KUKA KRL program: EPS_2_25369_MH2A_A_20251128065456.src

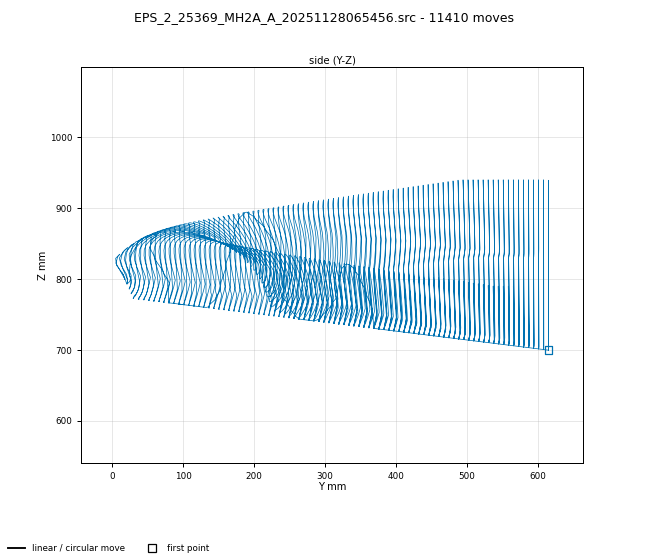
[picture p0: tool path of EPS_2_25369_MH2A_A_20251128065456.src, 11410 of 11412 moves have a stored position in this frame; points joined in program order, loops and branches not executed]
&ACCESS RVP
&REL 4
&COMMENT QRS 19112012
&PARAM EDITMASK = *
DEF PART()
EXT BAS (BAS_COMMAND :IN,REAL :IN )
INT I
BAS (#INITMOV,0 )

;KUKA QRS Post kuka4.cps  Date:22-06-2017 !

File_ID=2932

QRS_PRE_INIT()

;Init var - Until changes are made in qrs_pre_init
Outlet_Square_prg=0
Inlet_1_Square_prg=0
Inlet_2_Square_prg=0
Inlet_3_Square_prg=0
Inlet_4_Square_prg=0
Inlet_5_Square_prg=0

Outlet_1={X 0.000, Y 493.160, Z 839.500, B 0.000, E1 0.000 }
Inlet_1={X 0.000, Y 536.730, Z 239.500, B 0.000, E1 242.000 }
Outlet_1_type=201
Inlet_1_type=201
;QRS#1=Sidecore dimensions
;QRS#2=200-8" PVC SDR 35
;QRS#3=200-8" PVC SDR 35
;QRS#4=
;QRS#5=
;QRS#6=
;QRS#7=
;QRS#8=
;QRS#9=12-08 PSX
;QRS#10=12-08 PSX
;QRS#11=
;QRS#12=
;QRS#13=
;QRS#14=
;QRS#15=
;QRS#16=1220x127x1219 4'
;QRS#17=EPS Height
;QRS#18=940
;QRS#19=*
;QRS#20= UPDATED VERSION 22-06-2017
;QRS#21=*
Outlet_Square=0100
Inlet_1_Square=0100
Inlet_2_Square=0
Inlet_3_Square=0
Inlet_4_Square=0
Inlet_5_Square=0
Mill_Square=1
Outlet_Square_Prg=204
Inlet_1_Square_prg=204

QRS_INIT()

$ADVANCE=5

; T1
PTP {E1 173.443,E2 173.443}
PTP {X 0,Y 615.465,A -85,B 0,C 180,E1 173.443,E2 173.443,E3 0,E4 0,E5 0,E6 0}
QRS_SPEED_INIT()
LIN {X 0,Y 615.465,Z 699.696,A -85,B 0,C 180,E1 173.443,E2 173.443,E3 0,E4 0,E5 0,E6 0} C_VEL
LIN {X 0,Y 615.469,Z 699.697,A -85,B 0,C 180,E1 171.463,E2 171.463} C_VEL
LIN {X 0,Y 615.449,Z 699.694,A -85,B 0,C 180,E1 169.132,E2 169.132} C_VEL
LIN {X 0,Y 615.445,Z 699.691,A -85,B 0,C 180,E1 166.798,E2 166.798} C_VEL
LIN {X 0,Y 615.485,Z 699.687,A -85,B 0,C 180,E1 164.095,E2 164.095} C_VEL
LIN {X 0,Y 615.473,Z 699.698,A -85,B 0,C 180,E1 161.353,E2 161.353} C_VEL
LIN {X 0,Y 615.467,Z 699.698,A -85,B 0,C 180,E1 159.268,E2 159.268} C_VEL
LIN {X 0,Y 615.459,Z 699.697,A -85,B 0,C 180,E1 157.154,E2 157.154} C_VEL
LIN {X 0,Y 615.448,Z 699.697,A -85,B 0,C 180,E1 155.006,E2 155.006} C_VEL
LIN {X 0,Y 615.44,Z 699.696,A -85,B 0,C 180,E1 152.82,E2 152.82} C_VEL
LIN {X 0,Y 615.433,Z 699.695,A -85,B 0,C 180,E1 150.591,E2 150.591} C_VEL
LIN {X 0,Y 615.432,Z 699.694,A -85,B 0,C 180,E1 148.311,E2 148.311} C_VEL
LIN {X 0,Y 615.448,Z 699.692,A -85,B 0,C 180,E1 145.975,E2 145.975} C_VEL
LIN {X 0,Y 615.474,Z 699.699,A -85,B 0,C 180,E1 143.065,E2 143.065} C_VEL
LIN {X 0,Y 615.472,Z 699.697,A -85,B 0,C 180,E1 140.94,E2 140.94} C_VEL
LIN {X 0,Y 615.436,Z 699.696,A -85,B 0,C 180,E1 138.522,E2 138.522} C_VEL
LIN {X 0,Y 615.426,Z 699.695,A -85,B 0,C 180,E1 136.009,E2 136.009} C_VEL
LIN {X 0,Y 615.426,Z 699.695,A -85,B 0,C 180,E1 133.991,E2 133.991} C_VEL
LIN {X 0,Y 615.454,Z 699.695,A -85,B 0,C 180,E1 131.477,E2 131.477} C_VEL
LIN {X 0,Y 615.493,Z 699.698,A -85,B 0,C 180,E1 128.904,E2 128.904} C_VEL
LIN {X 0,Y 615.447,Z 699.695,A -85,B 0,C 180,E1 126.428,E2 126.428} C_VEL
LIN {X 0,Y 615.423,Z 699.696,A -85,B 0,C 180,E1 124.026,E2 124.026} C_VEL
LIN {X 0,Y 615.419,Z 699.697,A -85,B 0,C 180,E1 121.689,E2 121.689} C_VEL
LIN {X 0,Y 615.429,Z 699.698,A -85,B 0,C 180,E1 119.409,E2 119.409} C_VEL
LIN {X 0,Y 615.456,Z 699.7,A -85,B 0,C 180,E1 117.039,E2 117.039} C_VEL
LIN {X 0,Y 615.459,Z 699.694,A -85,B 0,C 180,E1 114.273,E2 114.273} C_VEL
LIN {X 0,Y 615.448,Z 699.694,A -85,B 0,C 180,E1 112.138,E2 112.138} C_VEL
LIN {X 0,Y 615.439,Z 699.695,A -85,B 0,C 180,E1 110.034,E2 110.034} C_VEL
LIN {X 0,Y 615.438,Z 699.695,A -85,B 0,C 180,E1 107.958,E2 107.958} C_VEL
LIN {X 0,Y 615.436,Z 699.695,A -85,B 0,C 180,E1 105.907,E2 105.907} C_VEL
LIN {X 0,Y 615.438,Z 699.695,A -85,B 0,C 180,E1 103.875,E2 103.875} C_VEL
LIN {X 0,Y 615.442,Z 699.694,A -85,B 0,C 180,E1 101.862,E2 101.862} C_VEL
LIN {X 0,Y 615.445,Z 699.694,A -85,B 0,C 180,E1 99.863,E2 99.863} C_VEL
LIN {X 0,Y 615.455,Z 699.692,A -85,B 0,C 180,E1 97.876,E2 97.876} C_VEL
LIN {X 0,Y 615.458,Z 699.693,A -85,B 0,C 180,E1 95.899,E2 95.899} C_VEL
LIN {X 0,Y 615.429,Z 699.694,A -85,B 0,C 180,E1 93.273,E2 93.273} C_VEL
LIN {X 0,Y 615.431,Z 699.694,A -85,B 0,C 180,E1 91.309,E2 91.309} C_VEL
LIN {X 0,Y 615.435,Z 699.693,A -85,B 0,C 180,E1 89.346,E2 89.346} C_VEL
LIN {X 0,Y 615.44,Z 699.692,A -85,B 0,C 180,E1 87.382,E2 87.382} C_VEL
LIN {X 0,Y 615.447,Z 699.691,A -85,B 0,C 180,E1 85.415,E2 85.415} C_VEL
LIN {X 0,Y 615.454,Z 699.69,A -85,B 0,C 180,E1 83.443,E2 83.443} C_VEL
LIN {X 0,Y 615.462,Z 699.689,A -85,B 0,C 180,E1 81.463,E2 81.463} C_VEL
LIN {X 0,Y 615.444,Z 699.691,A -85,B 0,C 180,E1 79.135,E2 79.135} C_VEL
LIN {X 0,Y 615.441,Z 699.693,A -85,B 0,C 180,E1 76.798,E2 76.798} C_VEL
LIN {X 0,Y 615.484,Z 699.701,A -85,B 0,C 180,E1 74.095,E2 74.095} C_VEL
LIN {X 0,Y 615.483,Z 699.685,A -85,B 0,C 180,E1 71.354,E2 71.354} C_VEL
LIN {X 0,Y 615.477,Z 699.686,A -85,B 0,C 180,E1 69.269,E2 69.269} C_VEL
LIN {X 0,Y 615.471,Z 699.686,A -85,B 0,C 180,E1 67.155,E2 67.155} C_VEL
LIN {X 0,Y 615.467,Z 699.686,A -85,B 0,C 180,E1 65.007,E2 65.007} C_VEL
LIN {X 0,Y 615.457,Z 699.688,A -85,B 0,C 180,E1 62.821,E2 62.821} C_VEL
LIN {X 0,Y 615.459,Z 699.695,A -85,B 0,C 180,E1 60.211,E2 60.211} C_VEL
LIN {X 0,Y 615.489,Z 699.695,A -85,B 0,C 180,E1 57.542,E2 57.542} C_VEL
LIN {X 0,Y 615.499,Z 699.684,A -85,B 0,C 180,E1 55.185,E2 55.185} C_VEL
LIN {X 0,Y 615.478,Z 699.683,A -85,B 0,C 180,E1 52.757,E2 52.757} C_VEL
LIN {X 0,Y 615.46,Z 699.69,A -85,B 0,C 180,E1 50.247,E2 50.247} C_VEL
LIN {X 0,Y 615.49,Z 699.699,A -85,B 0,C 180,E1 47.647,E2 47.647} C_VEL
LIN {X 0,Y 615.497,Z 699.683,A -85,B 0,C 180,E1 44.932,E2 44.932} C_VEL
LIN {X 0,Y 615.464,Z 699.69,A -85,B 0,C 180,E1 42.077,E2 42.077} C_VEL
LIN {X 0,Y 615.489,Z 699.696,A -85,B 0,C 180,E1 39.254,E2 39.254} C_VEL
LIN {X 0,Y 615.488,Z 714.003,A -85,B 0,C 180,E1 38.747,E2 38.747} C_VEL
LIN {X 0,Y 615.471,Z 726.147,A -85,B 0,C 180,E1 38.174,E2 38.174} C_VEL
LIN {X 0,Y 615.486,Z 736.877,A -85,B 0,C 180,E1 37.529,E2 37.529} C_VEL
LIN {X 0,Y 615.495,Z 746.56,A -85,B 0,C 180,E1 36.808,E2 36.808} C_VEL
LIN {X 0,Y 615.497,Z 755.612,A -85,B 0,C 180,E1 35.982,E2 35.982} C_VEL
LIN {X 0,Y 615.496,Z 764.246,A -85,B 0,C 180,E1 35.014,E2 35.014} C_VEL
LIN {X 0,Y 615.496,Z 771.392,A -85,B 0,C 180,E1 34.022,E2 34.022} C_VEL
LIN {X 0,Y 615.491,Z 775.986,A -85,B 0,C 180,E1 33.236,E2 33.236} C_VEL
LIN {X 0,Y 615.494,Z 781.677,A -85,B 0,C 180,E1 32.008,E2 32.008} C_VEL
LIN {X 0,Y 615.497,Z 785.306,A -85,B 0,C 180,E1 30.919,E2 30.919} C_VEL
LIN {X 0,Y 615.495,Z 787.813,A -85,B 0,C 180,E1 29.795,E2 29.795} C_VEL
LIN {X 0,Y 615.497,Z 789.275,A -85,B 0,C 180,E1 28.451,E2 28.451} C_VEL
LIN {X 0,Y 615.494,Z 789.086,A -85,B 0,C 180,E1 27.177,E2 27.177} C_VEL
LIN {X 0,Y 615.494,Z 788.342,A -85,B 0,C 180,E1 26.444,E2 26.444} C_VEL
LIN {X 0,Y 615.494,Z 786.748,A -85,B 0,C 180,E1 25.569,E2 25.569} C_VEL
LIN {X 0,Y 615.491,Z 784.237,A -85,B 0,C 180,E1 24.631,E2 24.631} C_VEL
LIN {X 0,Y 615.496,Z 780.239,A -85,B 0,C 180,E1 23.556,E2 23.556} C_VEL
LIN {X 0,Y 615.496,Z 775.556,A -85,B 0,C 180,E1 22.596,E2 22.596} C_VEL
LIN {X 0,Y 615.495,Z 769.504,A -85,B 0,C 180,E1 21.608,E2 21.608} C_VEL
LIN {X 0,Y 615.497,Z 761.465,A -85,B 0,C 180,E1 20.558,E2 20.558} C_VEL
LIN {X 0,Y 615.497,Z 753.124,A -85,B 0,C 180,E1 19.685,E2 19.685} C_VEL
LIN {X 0,Y 615.498,Z 742.968,A -85,B 0,C 180,E1 18.819,E2 18.819} C_VEL
LIN {X 0,Y 615.491,Z 732.83,A -85,B 0,C 180,E1 18.119,E2 18.119} C_VEL
LIN {X 0,Y 615.455,Z 722.15,A -85,B 0,C 180,E1 17.529,E2 17.529} C_VEL
LIN {X 0,Y 615.452,Z 710.214,A -85,B 0,C 180,E1 17.015,E2 17.015} C_VEL
LIN {X 0,Y 615.478,Z 699.698,A -85,B 0,C 180,E1 16.672,E2 16.672} C_VEL
LIN {X 0,Y 615.495,Z 699.683,A -85,B 0,C 180,E1 13.874,E2 13.874} C_VEL
LIN {X 0,Y 615.452,Z 699.69,A -85,B 0,C 180,E1 11.194,E2 11.194} C_VEL
LIN {X 0,Y 615.474,Z 699.698,A -85,B 0,C 180,E1 8.537,E2 8.537} C_VEL
LIN {X 0,Y 615.494,Z 699.688,A -85,B 0,C 180,E1 5.899,E2 5.899} C_VEL
LIN {X 0,Y 615.468,Z 699.685,A -85,B 0,C 180,E1 3.273,E2 3.273} C_VEL
LIN {X 0,Y 615.458,Z 699.694,A -85,B 0,C 180,E1 0.654,E2 0.654} C_VEL
LIN {X 0,Y 615.494,Z 699.697,A -85,B 0,C 180,E1 -1.963,E2 -1.963} C_VEL
LIN {X 0,Y 615.492,Z 699.682,A -85,B 0,C 180,E1 -4.584,E2 -4.584} C_VEL
LIN {X 0,Y 615.463,Z 699.688,A -85,B 0,C 180,E1 -7.216,E2 -7.216} C_VEL
LIN {X 0,Y 615.484,Z 699.698,A -85,B 0,C 180,E1 -9.862,E2 -9.862} C_VEL
LIN {X 0,Y 615.492,Z 699.686,A -85,B 0,C 180,E1 -12.53,E2 -12.53} C_VEL
LIN {X 0,Y 615.474,Z 699.684,A -85,B 0,C 180,E1 -15.226,E2 -15.226} C_VEL
LIN {X 0,Y 615.48,Z 699.697,A -85,B 0,C 180,E1 -17.957,E2 -17.957} C_VEL
LIN {X 0,Y 615.489,Z 699.686,A -85,B 0,C 180,E1 -20.731,E2 -20.731} C_VEL
LIN {X 0,Y 615.472,Z 699.686,A -85,B 0,C 180,E1 -23.557,E2 -23.557} C_VEL
LIN {X 0,Y 615.472,Z 699.688,A -85,B 0,C 180,E1 -25.716,E2 -25.716} C_VEL
LIN {X 0,Y 615.493,Z 699.698,A -85,B 0,C 180,E1 -28.45,E2 -28.45} C_VEL
LIN {X 0,Y 615.489,Z 699.683,A -85,B 0,C 180,E1 -31.086,E2 -31.086} C_VEL
LIN {X 0,Y 615.491,Z 699.68,A -85,B 0,C 180,E1 -33.534,E2 -33.534} C_VEL
LIN {X 0,Y 615.479,Z 699.686,A -85,B 0,C 180,E1 -35.832,E2 -35.832} C_VEL
LIN {X 0,Y 615.475,Z 699.69,A -85,B 0,C 180,E1 -38.07,E2 -38.07} C_VEL
LIN {X 0,Y 615.494,Z 699.7,A -85,B 0,C 180,E1 -40.606,E2 -40.606} C_VEL
LIN {X 0,Y 615.486,Z 699.685,A -85,B 0,C 180,E1 -43.245,E2 -43.245} C_VEL
LIN {X 0,Y 615.485,Z 699.684,A -85,B 0,C 180,E1 -46.003,E2 -46.003} C_VEL
LIN {X 0,Y 615.491,Z 699.695,A -85,B 0,C 180,E1 -48.905,E2 -48.905} C_VEL
LIN {X 0,Y 615.489,Z 699.691,A -85,B 0,C 180,E1 -51.095,E2 -51.095} C_VEL
LIN {X 0,Y 615.484,Z 699.683,A -85,B 0,C 180,E1 -53.575,E2 -53.575} C_VEL
LIN {X 0,Y 615.484,Z 699.799,A -85,B 0,C 180,E1 -54.356,E2 -54.356} C_VEL
LIN {X 0,Y 615.481,Z 713.626,A -85,B 0,C 180,E1 -57.153,E2 -57.153} C_VEL
LIN {X 0,Y 615.494,Z 727.321,A -85,B 0,C 180,E1 -59.84,E2 -59.84} C_VEL
LIN {X 0,Y 615.492,Z 741.016,A -85,B 0,C 180,E1 -62.454,E2 -62.454} C_VEL
LIN {X 0,Y 615.471,Z 754.706,A -85,B 0,C 180,E1 -65.007,E2 -65.007} C_VEL
LIN {X 0,Y 615.491,Z 769.177,A -85,B 0,C 180,E1 -67.654,E2 -67.654} C_VEL
LIN {X 0,Y 615.486,Z 784,A -85,B 0,C 180,E1 -70.315,E2 -70.315} C_VEL
LIN {X 0,Y 615.469,Z 799.609,A -85,B 0,C 180,E1 -73.071,E2 -73.071} C_VEL
LIN {X 0,Y 615.487,Z 815.037,A -85,B 0,C 180,E1 -75.761,E2 -75.761} C_VEL
LIN {X 0,Y 615.478,Z 829.932,A -85,B 0,C 180,E1 -78.327,E2 -78.327} C_VEL
LIN {X 0,Y 615.49,Z 843.234,A -85,B 0,C 180,E1 -78.557,E2 -78.557} C_VEL
LIN {X 0,Y 615.489,Z 856.372,A -85,B 0,C 180,E1 -78.923,E2 -78.923} C_VEL
LIN {X 0,Y 615.477,Z 868.148,A -85,B 0,C 180,E1 -79.384,E2 -79.384} C_VEL
LIN {X 0,Y 615.486,Z 879.573,A -85,B 0,C 180,E1 -79.972,E2 -79.972} C_VEL
LIN {X 0,Y 615.499,Z 891.019,A -85,B 0,C 180,E1 -80.718,E2 -80.718} C_VEL
LIN {X 0,Y 615.498,Z 900.256,A -85,B 0,C 180,E1 -81.463,E2 -81.463} C_VEL
LIN {X 0,Y 615.499,Z 908.652,A -85,B 0,C 180,E1 -82.29,E2 -82.29} C_VEL
LIN {X 0,Y 615.497,Z 916.69,A -85,B 0,C 180,E1 -83.259,E2 -83.259} C_VEL
LIN {X 0,Y 615.498,Z 922.422,A -85,B 0,C 180,E1 -84.101,E2 -84.101} C_VEL
LIN {X 0,Y 615.496,Z 927.872,A -85,B 0,C 180,E1 -85.087,E2 -85.087} C_VEL
LIN {X 0,Y 615.497,Z 932.141,A -85,B 0,C 180,E1 -86.071,E2 -86.071} C_VEL
LIN {X 0,Y 615.496,Z 934.398,A -85,B 0,C 180,E1 -86.727,E2 -86.727} C_VEL
LIN {X 0,Y 615.497,Z 936.233,A -85,B 0,C 180,E1 -87.382,E2 -87.382} C_VEL
LIN {X 0,Y 615.496,Z 937.608,A -85,B 0,C 180,E1 -88.037,E2 -88.037} C_VEL
LIN {X 0,Y 615.496,Z 939.173,A -85,B 0,C 180,E1 -89.346,E2 -89.346} C_VEL
LIN {X 0,Y 615.494,Z 939.389,A -85,B 0,C 180,E1 -90,E2 -90} C_VEL
LIN {X 0,Y 615.496,Z 938.58,A -85,B 0,C 180,E1 -91.309,E2 -91.309} C_VEL
LIN {X 0,Y 615.496,Z 937.608,A -85,B 0,C 180,E1 -91.963,E2 -91.963} C_VEL
LIN {X 0,Y 615.497,Z 936.233,A -85,B 0,C 180,E1 -92.618,E2 -92.618} C_VEL
LIN {X 0,Y 615.496,Z 933.35,A -85,B 0,C 180,E1 -93.601,E2 -93.601} C_VEL
LIN {X 0,Y 615.498,Z 929.442,A -85,B 0,C 180,E1 -94.584,E2 -94.584} C_VEL
LIN {X 0,Y 615.499,Z 924.405,A -85,B 0,C 180,E1 -95.57,E2 -95.57} C_VEL
LIN {X 0,Y 615.497,Z 917.869,A -85,B 0,C 180,E1 -96.583,E2 -96.583} C_VEL
LIN {X 0,Y 615.497,Z 910.133,A -85,B 0,C 180,E1 -97.545,E2 -97.545} C_VEL
LIN {X 0,Y 615.498,Z 902.045,A -85,B 0,C 180,E1 -98.371,E2 -98.371} C_VEL
LIN {X 0,Y 615.499,Z 892.168,A -85,B 0,C 180,E1 -99.199,E2 -99.199} C_VEL
LIN {X 0,Y 615.482,Z 880.983,A -85,B 0,C 180,E1 -99.945,E2 -99.945} C_VEL
LIN {X 0,Y 615.478,Z 870.024,A -85,B 0,C 180,E1 -100.527,E2 -100.527} C_VEL
LIN {X 0,Y 615.487,Z 857.564,A -85,B 0,C 180,E1 -101.037,E2 -101.037} C_VEL
LIN {X 0,Y 615.493,Z 845.064,A -85,B 0,C 180,E1 -101.401,E2 -101.401} C_VEL
LIN {X 0,Y 615.479,Z 831.469,A -85,B 0,C 180,E1 -101.652,E2 -101.652} C_VEL
LIN {X 0,Y 615.478,Z 829.797,A -85,B 0,C 180,E1 -101.694,E2 -101.694} C_VEL
LIN {X 0,Y 615.487,Z 815.037,A -85,B 0,C 180,E1 -104.239,E2 -104.239} C_VEL
LIN {X 0,Y 615.469,Z 799.61,A -85,B 0,C 180,E1 -106.929,E2 -106.929} C_VEL
LIN {X 0,Y 615.486,Z 784.001,A -85,B 0,C 180,E1 -109.685,E2 -109.685} C_VEL
LIN {X 0,Y 615.49,Z 767.803,A -85,B 0,C 180,E1 -112.595,E2 -112.595} C_VEL
LIN {X 0,Y 615.473,Z 753.141,A -85,B 0,C 180,E1 -115.282,E2 -115.282} C_VEL
LIN {X 0,Y 615.488,Z 739.06,A -85,B 0,C 180,E1 -117.915,E2 -117.915} C_VEL
LIN {X 0,Y 615.492,Z 725.365,A -85,B 0,C 180,E1 -120.539,E2 -120.539} C_VEL
LIN {X 0,Y 615.472,Z 711.67,A -85,B 0,C 180,E1 -123.237,E2 -123.237} C_VEL
LIN {X 0,Y 615.484,Z 699.687,A -85,B 0,C 180,E1 -125.671,E2 -125.671} C_VEL
LIN {X 0,Y 615.489,Z 699.681,A -85,B 0,C 180,E1 -128.069,E2 -128.069} C_VEL
LIN {X 0,Y 615.486,Z 699.684,A -85,B 0,C 180,E1 -130.607,E2 -130.607} C_VEL
LIN {X 0,Y 615.494,Z 699.699,A -85,B 0,C 180,E1 -133.244,E2 -133.244} C_VEL
LIN {X 0,Y 615.483,Z 699.685,A -85,B 0,C 180,E1 -136.003,E2 -136.003} C_VEL
LIN {X 0,Y 615.49,Z 699.686,A -85,B 0,C 180,E1 -138.905,E2 -138.905} C_VEL
LIN {X 0,Y 615.494,Z 699.689,A -85,B 0,C 180,E1 -141.096,E2 -141.096} C_VEL
LIN {X 0,Y 615.482,Z 699.7,A -85,B 0,C 180,E1 -143.575,E2 -143.575} C_VEL
LIN {X 0,Y 615.474,Z 699.691,A -85,B 0,C 180,E1 -145.977,E2 -145.977} C_VEL
LIN {X 0,Y 615.478,Z 699.685,A -85,B 0,C 180,E1 -148.314,E2 -148.314} C_VEL
LIN {X 0,Y 615.486,Z 699.681,A -85,B 0,C 180,E1 -150.594,E2 -150.594} C_VEL
LIN {X 0,Y 615.494,Z 699.697,A -85,B 0,C 180,E1 -153.556,E2 -153.556} C_VEL
LIN {X 0,Y 615.476,Z 699.695,A -85,B 0,C 180,E1 -155.995,E2 -155.995} C_VEL
LIN {X 0,Y 615.473,Z 699.685,A -85,B 0,C 180,E1 -158.568,E2 -158.568} C_VEL
LIN {X 0,Y 615.492,Z 699.688,A -85,B 0,C 180,E1 -161.395,E2 -161.395} C_VEL
LIN {X 0,Y 615.476,Z 699.696,A -85,B 0,C 180,E1 -164.095,E2 -164.095} C_VEL
LIN {X 0,Y 615.469,Z 699.685,A -85,B 0,C 180,E1 -166.798,E2 -166.798} C_VEL
LIN {X 0,Y 615.492,Z 699.686,A -85,B 0,C 180,E1 -169.473,E2 -169.473} C_VEL
LIN {X 0,Y 615.484,Z 699.698,A -85,B 0,C 180,E1 -172.124,E2 -172.124} C_VEL
LIN {X 0,Y 615.458,Z 699.689,A -85,B 0,C 180,E1 -174.759,E2 -174.759} C_VEL
LIN {X 0,Y 615.493,Z 699.682,A -85,B 0,C 180,E1 -177.382,E2 -177.382} C_VEL
LIN {X 0,Y 615.494,Z 699.697,A -85,B 0,C 180,E1 -180,E2 -180} C_VEL
LIN {X 0,Y 615.458,Z 699.694,A -85,B 0,C 180,E1 -182.618,E2 -182.618} C_VEL
LIN {X 0,Y 615.46,Z 699.687,A -85,B 0,C 180,E1 -185.242,E2 -185.242} C_VEL
LIN {X 0,Y 615.465,Z 699.696,A -85,B 0,C 180,E1 -186.557,E2 -186.557} C_VEL
LIN {X 0,Y 614.779,Z 699.837,A -85,B 0,C 180,E1 -187.103,E2 -187.103} C_VEL
LIN {X 0,Y 611.934,Z 700.259,A -85,B 0,C 180,E1 -187.99,E2 -187.99} C_VEL
LIN {X 0,Y 609.545,Z 700.565,A -85,B 0,C 180,E1 -188.702,E2 -188.702} C_VEL
LIN {X 0,Y 608.524,Z 700.679,A -85,B 0,C 180,E1 -189.252,E2 -189.252} C_VEL
LIN {X 0,Y 608.441,Z 700.688,A -85,B 0,C 180,E1 -189.438,E2 -189.438} C_VEL
LIN {X 0,Y 608.461,Z 700.691,A -85,B 0,C 180,E1 -192,E2 -192} C_VEL
LIN {X 0,Y 608.431,Z 700.694,A -85,B 0,C 180,E1 -194.722,E2 -194.722} C_VEL
LIN {X 0,Y 608.431,Z 700.694,A -85,B 0,C 180,E1 -196.785,E2 -196.785} C_VEL
LIN {X 0,Y 608.443,Z 700.692,A -85,B 0,C 180,E1 -198.87,E2 -198.87} C_VEL
LIN {X 0,Y 608.434,Z 700.692,A -85,B 0,C 180,E1 -200.982,E2 -200.982} C_VEL
LIN {X 0,Y 608.42,Z 700.693,A -85,B 0,C 180,E1 -203.125,E2 -203.125} C_VEL
LIN {X 0,Y 608.434,Z 700.689,A -85,B 0,C 180,E1 -205.713,E2 -205.713} C_VEL
LIN {X 0,Y 608.476,Z 700.695,A -85,B 0,C 180,E1 -208.62,E2 -208.62} C_VEL
LIN {X 0,Y 608.43,Z 700.691,A -85,B 0,C 180,E1 -211.319,E2 -211.319} C_VEL
LIN {X 0,Y 608.427,Z 700.69,A -85,B 0,C 180,E1 -213.728,E2 -213.728} C_VEL
LIN {X 0,Y 608.435,Z 700.69,A -85,B 0,C 180,E1 -216.093,E2 -216.093} C_VEL
LIN {X 0,Y 608.427,Z 700.697,A -85,B 0,C 180,E1 -218.592,E2 -218.592} C_VEL
LIN {X 0,Y 608.431,Z 700.692,A -85,B 0,C 180,E1 -221.339,E2 -221.339} C_VEL
LIN {X 0,Y 608.421,Z 700.691,A -85,B 0,C 180,E1 -223.874,E2 -223.874} C_VEL
LIN {X 0,Y 608.478,Z 700.69,A -85,B 0,C 180,E1 -226.691,E2 -226.691} C_VEL
LIN {X 0,Y 608.45,Z 700.696,A -85,B 0,C 180,E1 -228.823,E2 -228.823} C_VEL
LIN {X 0,Y 608.424,Z 700.691,A -85,B 0,C 180,E1 -231.765,E2 -231.765} C_VEL
LIN {X 0,Y 608.407,Z 700.693,A -85,B 0,C 180,E1 -233.96,E2 -233.96} C_VEL
LIN {X 0,Y 608.413,Z 700.692,A -85,B 0,C 180,E1 -236.326,E2 -236.326} C_VEL
LIN {X 0,Y 608.436,Z 700.693,A -85,B 0,C 180,E1 -238.735,E2 -238.735} C_VEL
LIN {X 0,Y 608.418,Z 700.693,A -85,B 0,C 180,E1 -241.732,E2 -241.732} C_VEL
LIN {X 0,Y 608.396,Z 700.694,A -85,B 0,C 180,E1 -244.295,E2 -244.295} C_VEL
LIN {X 0,Y 608.421,Z 700.695,A -85,B 0,C 180,E1 -246.875,E2 -246.875} C_VEL
LIN {X 0,Y 608.443,Z 700.692,A -85,B 0,C 180,E1 -249.725,E2 -249.725} C_VEL
LIN {X 0,Y 608.419,Z 700.694,A -85,B 0,C 180,E1 -251.827,E2 -251.827} C_VEL
LIN {X 0,Y 608.434,Z 700.692,A -85,B 0,C 180,E1 -253.905,E2 -253.905} C_VEL
LIN {X 0,Y 608.41,Z 700.692,A -85,B 0,C 180,E1 -256.642,E2 -256.642} C_VEL
LIN {X 0,Y 608.451,Z 700.695,A -85,B 0,C 180,E1 -259.35,E2 -259.35} C_VEL
LIN {X 0,Y 608.425,Z 700.693,A -85,B 0,C 180,E1 -262.032,E2 -262.032} C_VEL
LIN {X 0,Y 608.409,Z 700.692,A -85,B 0,C 180,E1 -264.698,E2 -264.698} C_VEL
LIN {X 0,Y 608.454,Z 700.692,A -85,B 0,C 180,E1 -267.352,E2 -267.352} C_VEL
LIN {X 0,Y 608.477,Z 700.689,A -85,B 0,C 180,E1 -270,E2 -270} C_VEL
LIN {X 0,Y 608.435,Z 700.689,A -85,B 0,C 180,E1 -272.648,E2 -272.648} C_VEL
LIN {X 0,Y 608.429,Z 700.693,A -85,B 0,C 180,E1 -275.302,E2 -275.302} C_VEL
LIN {X 0,Y 608.477,Z 700.693,A -85,B 0,C 180,E1 -277.967,E2 -277.967} C_VEL
LIN {X 0,Y 608.44,Z 700.689,A -85,B 0,C 180,E1 -280.65,E2 -280.65} C_VEL
LIN {X 0,Y 608.432,Z 700.691,A -85,B 0,C 180,E1 -283.357,E2 -283.357} C_VEL
LIN {X 0,Y 608.461,Z 700.695,A -85,B 0,C 180,E1 -286.094,E2 -286.094} C_VEL
LIN {X 0,Y 608.448,Z 700.687,A -85,B 0,C 180,E1 -288.87,E2 -288.87} C_VEL
LIN {X 0,Y 608.442,Z 700.688,A -85,B 0,C 180,E1 -290.982,E2 -290.982} C_VEL
LIN {X 0,Y 608.43,Z 700.689,A -85,B 0,C 180,E1 -293.125,E2 -293.125} C_VEL
LIN {X 0,Y 608.448,Z 700.691,A -85,B 0,C 180,E1 -295.715,E2 -295.715} C_VEL
LIN {X 0,Y 608.481,Z 700.687,A -85,B 0,C 180,E1 -298.621,E2 -298.621} C_VEL
LIN {X 0,Y 608.441,Z 700.688,A -85,B 0,C 180,E1 -301.318,E2 -301.318} C_VEL
LIN {X 0,Y 608.428,Z 700.692,A -85,B 0,C 180,E1 -303.728,E2 -303.728} C_VEL
LIN {X 0,Y 608.444,Z 700.695,A -85,B 0,C 180,E1 -306.093,E2 -306.093} C_VEL
LIN {X 0,Y 608.472,Z 700.692,A -85,B 0,C 180,E1 -308.588,E2 -308.588} C_VEL
LIN {X 0,Y 608.455,Z 700.686,A -85,B 0,C 180,E1 -311.341,E2 -311.341} C_VEL
LIN {X 0,Y 608.456,Z 700.688,A -85,B 0,C 180,E1 -313.871,E2 -313.871} C_VEL
LIN {X 0,Y 608.477,Z 700.692,A -85,B 0,C 180,E1 -316.691,E2 -316.691} C_VEL
LIN {X 0,Y 608.457,Z 700.686,A -85,B 0,C 180,E1 -319.697,E2 -319.697} C_VEL
LIN {X 0,Y 608.465,Z 700.696,A -85,B 0,C 180,E1 -320.654,E2 -320.654} C_VEL
LIN {X 0,Y 608.503,Z 713.389,A -85,B 0,C 180,E1 -321.096,E2 -321.096} C_VEL
LIN {X 0,Y 608.485,Z 724.662,A -85,B 0,C 180,E1 -321.619,E2 -321.619} C_VEL
LIN {X 0,Y 608.472,Z 736.703,A -85,B 0,C 180,E1 -322.335,E2 -322.335} C_VEL
LIN {X 0,Y 608.467,Z 746.782,A -85,B 0,C 180,E1 -323.086,E2 -323.086} C_VEL
LIN {X 0,Y 608.455,Z 756.207,A -85,B 0,C 180,E1 -323.954,E2 -323.954} C_VEL
LIN {X 0,Y 608.467,Z 764.899,A -85,B 0,C 180,E1 -324.938,E2 -324.938} C_VEL
LIN {X 0,Y 608.441,Z 771.955,A -85,B 0,C 180,E1 -325.928,E2 -325.928} C_VEL
LIN {X 0,Y 608.43,Z 778.577,A -85,B 0,C 180,E1 -327.119,E2 -327.119} C_VEL
LIN {X 0,Y 608.428,Z 783.503,A -85,B 0,C 180,E1 -328.293,E2 -328.293} C_VEL
LIN {X 0,Y 608.433,Z 786.942,A -85,B 0,C 180,E1 -329.453,E2 -329.453} C_VEL
LIN {X 0,Y 608.445,Z 788.467,A -85,B 0,C 180,E1 -330.219,E2 -330.219} C_VEL
LIN {X 0,Y 608.421,Z 789.788,A -85,B 0,C 180,E1 -331.39,E2 -331.39} C_VEL
LIN {X 0,Y 608.436,Z 789.717,A -85,B 0,C 180,E1 -332.801,E2 -332.801} C_VEL
LIN {X 0,Y 608.421,Z 788.314,A -85,B 0,C 180,E1 -333.963,E2 -333.963} C_VEL
LIN {X 0,Y 608.433,Z 785.822,A -85,B 0,C 180,E1 -335.063,E2 -335.063} C_VEL
LIN {X 0,Y 608.441,Z 782.175,A -85,B 0,C 180,E1 -336.154,E2 -336.154} C_VEL
LIN {X 0,Y 608.447,Z 777.282,A -85,B 0,C 180,E1 -337.235,E2 -337.235} C_VEL
LIN {X 0,Y 608.438,Z 770.991,A -85,B 0,C 180,E1 -338.307,E2 -338.307} C_VEL
LIN {X 0,Y 608.458,Z 763.49,A -85,B 0,C 180,E1 -339.325,E2 -339.325} C_VEL
LIN {X 0,Y 608.477,Z 755.053,A -85,B 0,C 180,E1 -340.254,E2 -340.254} C_VEL
LIN {X 0,Y 608.472,Z 745.197,A -85,B 0,C 180,E1 -341.131,E2 -341.131} C_VEL
LIN {X 0,Y 608.507,Z 734.234,A -85,B 0,C 180,E1 -341.917,E2 -341.917} C_VEL
LIN {X 0,Y 608.481,Z 723.664,A -85,B 0,C 180,E1 -342.524,E2 -342.524} C_VEL
LIN {X 0,Y 608.472,Z 712.168,A -85,B 0,C 180,E1 -343.043,E2 -343.043} C_VEL
LIN {X 0,Y 608.472,Z 700.695,A -85,B 0,C 180,E1 -343.446,E2 -343.446} C_VEL
LIN {X 0,Y 608.481,Z 700.687,A -85,B 0,C 180,E1 -345.98,E2 -345.98} C_VEL
LIN {X 0,Y 608.429,Z 700.69,A -85,B 0,C 180,E1 -348.675,E2 -348.675} C_VEL
LIN {X 0,Y 608.443,Z 700.694,A -85,B 0,C 180,E1 -351.364,E2 -351.364} C_VEL
LIN {X 0,Y 608.466,Z 700.69,A -85,B 0,C 180,E1 -354.033,E2 -354.033} C_VEL
LIN {X 0,Y 608.465,Z 700.685,A -85,B 0,C 180,E1 -356.689,E2 -356.689} C_VEL
LIN {X 0,Y 608.456,Z 700.69,A -85,B 0,C 180,E1 -359.338,E2 -359.338} C_VEL
LIN {X 0,Y 608.464,Z 700.694,A -85,B 0,C 180,E1 -361.986,E2 -361.986} C_VEL
LIN {X 0,Y 608.459,Z 700.687,A -85,B 0,C 180,E1 -364.638,E2 -364.638} C_VEL
LIN {X 0,Y 608.435,Z 700.69,A -85,B 0,C 180,E1 -367.3,E2 -367.3} C_VEL
LIN {X 0,Y 608.456,Z 700.697,A -85,B 0,C 180,E1 -369.977,E2 -369.977} C_VEL
LIN {X 0,Y 608.477,Z 700.685,A -85,B 0,C 180,E1 -372.677,E2 -372.677} C_VEL
LIN {X 0,Y 608.462,Z 700.686,A -85,B 0,C 180,E1 -375.406,E2 -375.406} C_VEL
LIN {X 0,Y 608.448,Z 700.699,A -85,B 0,C 180,E1 -378.172,E2 -378.172} C_VEL
LIN {X 0,Y 608.455,Z 700.687,A -85,B 0,C 180,E1 -380.982,E2 -380.982} C_VEL
LIN {X 0,Y 608.449,Z 700.687,A -85,B 0,C 180,E1 -383.124,E2 -383.124} C_VEL
LIN {X 0,Y 608.462,Z 700.688,A -85,B 0,C 180,E1 -385.718,E2 -385.718} C_VEL
LIN {X 0,Y 608.452,Z 700.697,A -85,B 0,C 180,E1 -388.267,E2 -388.267} C_VEL
LIN {X 0,Y 608.471,Z 700.693,A -85,B 0,C 180,E1 -390.545,E2 -390.545} C_VEL
LIN {X 0,Y 608.464,Z 700.689,A -85,B 0,C 180,E1 -392.879,E2 -392.879} C_VEL
LIN {X 0,Y 608.45,Z 700.687,A -85,B 0,C 180,E1 -395.277,E2 -395.277} C_VEL
LIN {X 0,Y 608.464,Z 700.686,A -85,B 0,C 180,E1 -397.747,E2 -397.747} C_VEL
LIN {X 0,Y 608.45,Z 700.694,A -85,B 0,C 180,E1 -400.328,E2 -400.328} C_VEL
LIN {X 0,Y 608.474,Z 700.685,A -85,B 0,C 180,E1 -403.309,E2 -403.309} C_VEL
LIN {X 0,Y 608.472,Z 700.687,A -85,B 0,C 180,E1 -406.13,E2 -406.13} C_VEL
LIN {X 0,Y 608.46,Z 700.696,A -85,B 0,C 180,E1 -408.823,E2 -408.823} C_VEL
LIN {X 0,Y 608.47,Z 700.685,A -85,B 0,C 180,E1 -411.76,E2 -411.76} C_VEL
LIN {X 0,Y 608.492,Z 700.74,A -85,B 0,C 180,E1 -414.08,E2 -414.08} C_VEL
LIN {X 0,Y 608.676,Z 706.578,A -85,B 0,C 180,E1 -415.302,E2 -415.302} C_VEL
LIN {X 0,Y 608.66,Z 719.495,A -85,B 0,C 180,E1 -417.917,E2 -417.917} C_VEL
LIN {X 0,Y 608.596,Z 733.19,A -85,B 0,C 180,E1 -420.608,E2 -420.608} C_VEL
LIN {X 0,Y 608.57,Z 746.885,A -85,B 0,C 180,E1 -423.231,E2 -423.231} C_VEL
LIN {X 0,Y 608.54,Z 760.792,A -85,B 0,C 180,E1 -425.835,E2 -425.835} C_VEL
LIN {X 0,Y 608.528,Z 776.232,A -85,B 0,C 180,E1 -428.666,E2 -428.666} C_VEL
LIN {X 0,Y 608.493,Z 792.297,A -85,B 0,C 180,E1 -431.555,E2 -431.555} C_VEL
LIN {X 0,Y 608.481,Z 807.534,A -85,B 0,C 180,E1 -434.251,E2 -434.251} C_VEL
LIN {X 0,Y 608.459,Z 823.186,A -85,B 0,C 180,E1 -436.983,E2 -436.983} C_VEL
LIN {X 0,Y 608.439,Z 830.156,A -85,B 0,C 180,E1 -438.19,E2 -438.19} C_VEL
LIN {X 0,Y 608.54,Z 844.261,A -85,B 0,C 180,E1 -438.445,E2 -438.445} C_VEL
LIN {X 0,Y 608.531,Z 856.957,A -85,B 0,C 180,E1 -438.81,E2 -438.81} C_VEL
LIN {X 0,Y 608.499,Z 868.679,A -85,B 0,C 180,E1 -439.279,E2 -439.279} C_VEL
LIN {X 0,Y 608.482,Z 879.753,A -85,B 0,C 180,E1 -439.855,E2 -439.855} C_VEL
LIN {X 0,Y 608.504,Z 891.25,A -85,B 0,C 180,E1 -440.611,E2 -440.611} C_VEL
LIN {X 0,Y 608.472,Z 900.535,A -85,B 0,C 180,E1 -441.364,E2 -441.364} C_VEL
LIN {X 0,Y 608.456,Z 908.988,A -85,B 0,C 180,E1 -442.2,E2 -442.2} C_VEL
LIN {X 0,Y 608.462,Z 917.234,A -85,B 0,C 180,E1 -443.201,E2 -443.201} C_VEL
LIN {X 0,Y 608.437,Z 923.876,A -85,B 0,C 180,E1 -444.199,E2 -444.199} C_VEL
LIN {X 0,Y 608.432,Z 929.95,A -85,B 0,C 180,E1 -445.362,E2 -445.362} C_VEL
LIN {X 0,Y 608.449,Z 933.896,A -85,B 0,C 180,E1 -446.358,E2 -446.358} C_VEL
LIN {X 0,Y 608.425,Z 936.809,A -85,B 0,C 180,E1 -447.352,E2 -447.352} C_VEL
LIN {X 0,Y 608.441,Z 938.201,A -85,B 0,C 180,E1 -448.014,E2 -448.014} C_VEL
LIN {X 0,Y 608.438,Z 939.783,A -85,B 0,C 180,E1 -449.338,E2 -449.338} C_VEL
LIN {X 0,Y 608.434,Z 940,A -85,B 0,C 180,E1 -450,E2 -450} C_VEL
LIN {X 0,Y 608.448,Z 939.184,A -85,B 0,C 180,E1 -451.324,E2 -451.324} C_VEL
LIN {X 0,Y 608.441,Z 938.201,A -85,B 0,C 180,E1 -451.986,E2 -451.986} C_VEL
LIN {X 0,Y 608.425,Z 936.809,A -85,B 0,C 180,E1 -452.648,E2 -452.648} C_VEL
LIN {X 0,Y 608.449,Z 933.896,A -85,B 0,C 180,E1 -453.642,E2 -453.642} C_VEL
LIN {X 0,Y 608.432,Z 929.95,A -85,B 0,C 180,E1 -454.638,E2 -454.638} C_VEL
LIN {X 0,Y 608.437,Z 923.877,A -85,B 0,C 180,E1 -455.801,E2 -455.801} C_VEL
LIN {X 0,Y 608.462,Z 917.235,A -85,B 0,C 180,E1 -456.799,E2 -456.799} C_VEL
LIN {X 0,Y 608.456,Z 908.989,A -85,B 0,C 180,E1 -457.8,E2 -457.8} C_VEL
LIN {X 0,Y 608.472,Z 900.536,A -85,B 0,C 180,E1 -458.636,E2 -458.636} C_VEL
LIN {X 0,Y 608.48,Z 890.091,A -85,B 0,C 180,E1 -459.473,E2 -459.473} C_VEL
LIN {X 0,Y 608.482,Z 879.755,A -85,B 0,C 180,E1 -460.145,E2 -460.145} C_VEL
LIN {X 0,Y 608.497,Z 868.296,A -85,B 0,C 180,E1 -460.739,E2 -460.739} C_VEL
LIN {X 0,Y 608.538,Z 855.949,A -85,B 0,C 180,E1 -461.223,E2 -461.223} C_VEL
LIN {X 0,Y 608.538,Z 842.439,A -85,B 0,C 180,E1 -461.597,E2 -461.597} C_VEL
LIN {X 0,Y 608.439,Z 830.157,A -85,B 0,C 180,E1 -461.81,E2 -461.81} C_VEL
LIN {X 0,Y 608.464,Z 815.361,A -85,B 0,C 180,E1 -464.379,E2 -464.379} C_VEL
LIN {X 0,Y 608.468,Z 799.71,A -85,B 0,C 180,E1 -467.13,E2 -467.13} C_VEL
LIN {X 0,Y 608.508,Z 784.058,A -85,B 0,C 180,E1 -469.92,E2 -469.92} C_VEL
LIN {X 0,Y 608.539,Z 768.409,A -85,B 0,C 180,E1 -472.761,E2 -472.761} C_VEL
LIN {X 0,Y 608.57,Z 753.525,A -85,B 0,C 180,E1 -475.518,E2 -475.518} C_VEL
LIN {X 0,Y 608.585,Z 739.06,A -85,B 0,C 180,E1 -478.26,E2 -478.26} C_VEL
LIN {X 0,Y 608.604,Z 725.405,A -85,B 0,C 180,E1 -480.914,E2 -480.914} C_VEL
LIN {X 0,Y 608.641,Z 713.627,A -85,B 0,C 180,E1 -483.263,E2 -483.263} C_VEL
LIN {X 0,Y 608.693,Z 701.985,A -85,B 0,C 180,E1 -485.647,E2 -485.647} C_VEL
LIN {X 0,Y 608.466,Z 700.688,A -85,B 0,C 180,E1 -485.986,E2 -485.986} C_VEL
LIN {X 0,Y 608.472,Z 700.686,A -85,B 0,C 180,E1 -488.588,E2 -488.588} C_VEL
LIN {X 0,Y 608.465,Z 700.695,A -85,B 0,C 180,E1 -491.342,E2 -491.342} C_VEL
LIN {X 0,Y 608.463,Z 700.685,A -85,B 0,C 180,E1 -494.264,E2 -494.264} C_VEL
LIN {X 0,Y 608.458,Z 700.691,A -85,B 0,C 180,E1 -497.04,E2 -497.04} C_VEL
LIN {X 0,Y 608.455,Z 700.692,A -85,B 0,C 180,E1 -499.697,E2 -499.697} C_VEL
LIN {X 0,Y 608.464,Z 700.686,A -85,B 0,C 180,E1 -502.253,E2 -502.253} C_VEL
LIN {X 0,Y 608.487,Z 700.686,A -85,B 0,C 180,E1 -505.09,E2 -505.09} C_VEL
LIN {X 0,Y 608.467,Z 700.69,A -85,B 0,C 180,E1 -507.906,E2 -507.906} C_VEL
LIN {X 0,Y 608.458,Z 700.688,A -85,B 0,C 180,E1 -510.22,E2 -510.22} C_VEL
LIN {X 0,Y 608.482,Z 700.683,A -85,B 0,C 180,E1 -512.793,E2 -512.793} C_VEL
LIN {X 0,Y 608.474,Z 700.692,A -85,B 0,C 180,E1 -515.849,E2 -515.849} C_VEL
LIN {X 0,Y 608.461,Z 700.688,A -85,B 0,C 180,E1 -518.308,E2 -518.308} C_VEL
LIN {X 0,Y 608.457,Z 700.687,A -85,B 0,C 180,E1 -521.13,E2 -521.13} C_VEL
LIN {X 0,Y 608.458,Z 700.696,A -85,B 0,C 180,E1 -523.906,E2 -523.906} C_VEL
LIN {X 0,Y 608.448,Z 700.688,A -85,B 0,C 180,E1 -526.643,E2 -526.643} C_VEL
LIN {X 0,Y 608.468,Z 700.687,A -85,B 0,C 180,E1 -529.35,E2 -529.35} C_VEL
LIN {X 0,Y 608.478,Z 700.694,A -85,B 0,C 180,E1 -532.033,E2 -532.033} C_VEL
LIN {X 0,Y 608.442,Z 700.689,A -85,B 0,C 180,E1 -534.698,E2 -534.698} C_VEL
LIN {X 0,Y 608.482,Z 700.684,A -85,B 0,C 180,E1 -537.352,E2 -537.352} C_VEL
LIN {X 0,Y 608.484,Z 700.692,A -85,B 0,C 180,E1 -540,E2 -540} C_VEL
LIN {X 0,Y 608.452,Z 700.69,A -85,B 0,C 180,E1 -542.648,E2 -542.648} C_VEL
LIN {X 0,Y 608.444,Z 700.688,A -85,B 0,C 180,E1 -545.302,E2 -545.302} C_VEL
LIN {X 0,Y 608.483,Z 700.689,A -85,B 0,C 180,E1 -547.967,E2 -547.967} C_VEL
LIN {X 0,Y 608.441,Z 700.688,A -85,B 0,C 180,E1 -549.438,E2 -549.438} C_VEL
LIN {X 0,Y 607.781,Z 700.778,A -85,B 0,C 180,E1 -549.991,E2 -549.991} C_VEL
LIN {X 0,Y 604.939,Z 701.133,A -85,B 0,C 180,E1 -550.887,E2 -550.887} C_VEL
LIN {X 0,Y 602.531,Z 701.434,A -85,B 0,C 180,E1 -551.609,E2 -551.609} C_VEL
LIN {X 0,Y 601.49,Z 701.562,A -85,B 0,C 180,E1 -552.165,E2 -552.165} C_VEL
LIN {X 0,Y 601.402,Z 701.57,A -85,B 0,C 180,E1 -552.354,E2 -552.354} C_VEL
LIN {X 0,Y 601.396,Z 701.569,A -85,B 0,C 180,E1 -554.898,E2 -554.898} C_VEL
LIN {X 0,Y 601.403,Z 701.567,A -85,B 0,C 180,E1 -556.987,E2 -556.987} C_VEL
LIN {X 0,Y 601.392,Z 701.568,A -85,B 0,C 180,E1 -559.81,E2 -559.81} C_VEL
LIN {X 0,Y 601.418,Z 701.573,A -85,B 0,C 180,E1 -562.605,E2 -562.605} C_VEL
LIN {X 0,Y 601.38,Z 701.573,A -85,B 0,C 180,E1 -564.88,E2 -564.88} C_VEL
LIN {X 0,Y 601.374,Z 701.569,A -85,B 0,C 180,E1 -567.354,E2 -567.354} C_VEL
LIN {X 0,Y 601.378,Z 701.569,A -85,B 0,C 180,E1 -569.396,E2 -569.396} C_VEL
LIN {X 0,Y 601.39,Z 701.567,A -85,B 0,C 180,E1 -571.728,E2 -571.728} C_VEL
LIN {X 0,Y 601.412,Z 701.566,A -85,B 0,C 180,E1 -574.12,E2 -574.12} C_VEL
LIN {X 0,Y 601.394,Z 701.574,A -85,B 0,C 180,E1 -576.584,E2 -576.584} C_VEL
LIN {X 0,Y 601.389,Z 701.568,A -85,B 0,C 180,E1 -579.529,E2 -579.529} C_VEL
LIN {X 0,Y 601.395,Z 701.566,A -85,B 0,C 180,E1 -581.768,E2 -581.768} C_VEL
LIN {X 0,Y 601.401,Z 701.57,A -85,B 0,C 180,E1 -584.533,E2 -584.533} C_VEL
LIN {X 0,Y 601.369,Z 701.573,A -85,B 0,C 180,E1 -587.414,E2 -587.414} C_VEL
LIN {X 0,Y 601.376,Z 701.568,A -85,B 0,C 180,E1 -590.002,E2 -590.002} C_VEL
LIN {X 0,Y 601.4,Z 701.569,A -85,B 0,C 180,E1 -592.623,E2 -592.623} C_VEL
LIN {X 0,Y 601.413,Z 701.575,A -85,B 0,C 180,E1 -595.068,E2 -595.068} C_VEL
LIN {X 0,Y 601.411,Z 701.569,A -85,B 0,C 180,E1 -597.483,E2 -597.483} C_VEL
LIN {X 0,Y 601.371,Z 701.57,A -85,B 0,C 180,E1 -599.862,E2 -599.862} C_VEL
LIN {X 0,Y 601.354,Z 701.571,A -85,B 0,C 180,E1 -602.129,E2 -602.129} C_VEL
LIN {X 0,Y 601.352,Z 701.572,A -85,B 0,C 180,E1 -604.379,E2 -604.379} C_VEL
LIN {X 0,Y 601.361,Z 701.571,A -85,B 0,C 180,E1 -606.587,E2 -606.587} C_VEL
LIN {X 0,Y 601.427,Z 701.571,A -85,B 0,C 180,E1 -609.478,E2 -609.478} C_VEL
LIN {X 0,Y 601.39,Z 701.573,A -85,B 0,C 180,E1 -611.607,E2 -611.607} C_VEL
LIN {X 0,Y 601.429,Z 701.568,A -85,B 0,C 180,E1 -613.713,E2 -613.713} C_VEL
LIN {X 0,Y 601.371,Z 701.569,A -85,B 0,C 180,E1 -616.483,E2 -616.483} C_VEL
LIN {X 0,Y 601.385,Z 701.573,A -85,B 0,C 180,E1 -619.223,E2 -619.223} C_VEL
LIN {X 0,Y 601.401,Z 701.57,A -85,B 0,C 180,E1 -621.939,E2 -621.939} C_VEL
LIN {X 0,Y 601.378,Z 701.568,A -85,B 0,C 180,E1 -624.636,E2 -624.636} C_VEL
LIN {X 0,Y 601.419,Z 701.568,A -85,B 0,C 180,E1 -627.321,E2 -627.321} C_VEL
LIN {X 0,Y 601.445,Z 701.565,A -85,B 0,C 180,E1 -630,E2 -630} C_VEL
LIN {X 0,Y 601.403,Z 701.565,A -85,B 0,C 180,E1 -632.679,E2 -632.679} C_VEL
LIN {X 0,Y 601.398,Z 701.569,A -85,B 0,C 180,E1 -635.364,E2 -635.364} C_VEL
LIN {X 0,Y 601.438,Z 701.568,A -85,B 0,C 180,E1 -638.061,E2 -638.061} C_VEL
LIN {X 0,Y 601.393,Z 701.566,A -85,B 0,C 180,E1 -640.994,E2 -640.994} C_VEL
LIN {X 0,Y 601.397,Z 701.57,A -85,B 0,C 180,E1 -643.516,E2 -643.516} C_VEL
LIN {X 0,Y 601.442,Z 701.566,A -85,B 0,C 180,E1 -646.287,E2 -646.287} C_VEL
LIN {X 0,Y 601.41,Z 701.564,A -85,B 0,C 180,E1 -649.099,E2 -649.099} C_VEL
LIN {X 0,Y 601.395,Z 701.566,A -85,B 0,C 180,E1 -651.24,E2 -651.24} C_VEL
LIN {X 0,Y 601.459,Z 701.569,A -85,B 0,C 180,E1 -654.14,E2 -654.14} C_VEL
LIN {X 0,Y 601.4,Z 701.565,A -85,B 0,C 180,E1 -657.114,E2 -657.114} C_VEL
LIN {X 0,Y 601.405,Z 701.565,A -85,B 0,C 180,E1 -659.394,E2 -659.394} C_VEL
LIN {X 0,Y 601.4,Z 701.568,A -85,B 0,C 180,E1 -661.727,E2 -661.727} C_VEL
LIN {X 0,Y 601.416,Z 701.571,A -85,B 0,C 180,E1 -664.119,E2 -664.119} C_VEL
LIN {X 0,Y 601.437,Z 701.561,A -85,B 0,C 180,E1 -667.382,E2 -667.382} C_VEL
LIN {X 0,Y 601.403,Z 701.569,A -85,B 0,C 180,E1 -669.996,E2 -669.996} C_VEL
LIN {X 0,Y 601.418,Z 701.57,A -85,B 0,C 180,E1 -672.67,E2 -672.67} C_VEL
LIN {X 0,Y 601.403,Z 701.565,A -85,B 0,C 180,E1 -675.479,E2 -675.479} C_VEL
LIN {X 0,Y 601.425,Z 701.571,A -85,B 0,C 180,E1 -678.407,E2 -678.407} C_VEL
LIN {X 0,Y 601.44,Z 701.572,A -85,B 0,C 180,E1 -680.545,E2 -680.545} C_VEL
LIN {X 0,Y 601.53,Z 713.447,A -85,B 0,C 180,E1 -680.971,E2 -680.971} C_VEL
LIN {X 0,Y 601.476,Z 725.185,A -85,B 0,C 180,E1 -681.524,E2 -681.524} C_VEL
LIN {X 0,Y 601.462,Z 737.385,A -85,B 0,C 180,E1 -682.266,E2 -682.266} C_VEL
LIN {X 0,Y 601.453,Z 748.235,A -85,B 0,C 180,E1 -683.107,E2 -683.107} C_VEL
LIN {X 0,Y 601.418,Z 756.46,A -85,B 0,C 180,E1 -683.885,E2 -683.885} C_VEL
LIN {X 0,Y 601.391,Z 765.168,A -85,B 0,C 180,E1 -684.889,E2 -684.889} C_VEL
LIN {X 0,Y 601.378,Z 772.089,A -85,B 0,C 180,E1 -685.878,E2 -685.878} C_VEL
LIN {X 0,Y 601.348,Z 778.363,A -85,B 0,C 180,E1 -687.015,E2 -687.015} C_VEL
LIN {X 0,Y 601.345,Z 783.582,A -85,B 0,C 180,E1 -688.269,E2 -688.269} C_VEL
LIN {X 0,Y 601.319,Z 785.986,A -85,B 0,C 180,E1 -689.052,E2 -689.052} C_VEL
LIN {X 0,Y 601.35,Z 787.889,A -85,B 0,C 180,E1 -689.865,E2 -689.865} C_VEL
LIN {X 0,Y 601.338,Z 789.063,A -85,B 0,C 180,E1 -690.602,E2 -690.602} C_VEL
LIN {X 0,Y 601.33,Z 789.779,A -85,B 0,C 180,E1 -691.368,E2 -691.368} C_VEL
LIN {X 0,Y 601.352,Z 789.828,A -85,B 0,C 180,E1 -692.65,E2 -692.65} C_VEL
LIN {X 0,Y 601.317,Z 788.878,A -85,B 0,C 180,E1 -693.632,E2 -693.632} C_VEL
LIN {X 0,Y 601.333,Z 787.562,A -85,B 0,C 180,E1 -694.378,E2 -694.378} C_VEL
LIN {X 0,Y 601.344,Z 785.772,A -85,B 0,C 180,E1 -695.119,E2 -695.119} C_VEL
LIN {X 0,Y 601.344,Z 782.108,A -85,B 0,C 180,E1 -696.221,E2 -696.221} C_VEL
LIN {X 0,Y 601.372,Z 776.691,A -85,B 0,C 180,E1 -697.406,E2 -697.406} C_VEL
LIN {X 0,Y 601.364,Z 770.864,A -85,B 0,C 180,E1 -698.399,E2 -698.399} C_VEL
LIN {X 0,Y 601.387,Z 762.958,A -85,B 0,C 180,E1 -699.476,E2 -699.476} C_VEL
LIN {X 0,Y 601.413,Z 754.886,A -85,B 0,C 180,E1 -700.368,E2 -700.368} C_VEL
LIN {X 0,Y 601.431,Z 744.861,A -85,B 0,C 180,E1 -701.265,E2 -701.265} C_VEL
LIN {X 0,Y 601.489,Z 733.968,A -85,B 0,C 180,E1 -702.051,E2 -702.051} C_VEL
LIN {X 0,Y 601.479,Z 723.306,A -85,B 0,C 180,E1 -702.665,E2 -702.665} C_VEL
LIN {X 0,Y 601.515,Z 711.677,A -85,B 0,C 180,E1 -703.191,E2 -703.191} C_VEL
LIN {X 0,Y 601.448,Z 701.571,A -85,B 0,C 180,E1 -703.553,E2 -703.553} C_VEL
LIN {X 0,Y 601.403,Z 701.565,A -85,B 0,C 180,E1 -706.484,E2 -706.484} C_VEL
LIN {X 0,Y 601.393,Z 701.571,A -85,B 0,C 180,E1 -709.223,E2 -709.223} C_VEL
LIN {X 0,Y 601.443,Z 701.566,A -85,B 0,C 180,E1 -711.939,E2 -711.939} C_VEL
LIN {X 0,Y 601.413,Z 701.564,A -85,B 0,C 180,E1 -714.636,E2 -714.636} C_VEL
LIN {X 0,Y 601.425,Z 701.566,A -85,B 0,C 180,E1 -717.321,E2 -717.321} C_VEL
LIN {X 0,Y 601.453,Z 701.567,A -85,B 0,C 180,E1 -720,E2 -720} C_VEL
LIN {X 0,Y 601.447,Z 701.56,A -85,B 0,C 180,E1 -722.679,E2 -722.679} C_VEL
LIN {X 0,Y 601.412,Z 701.566,A -85,B 0,C 180,E1 -725.364,E2 -725.364} C_VEL
LIN {X 0,Y 601.442,Z 701.569,A -85,B 0,C 180,E1 -728.061,E2 -728.061} C_VEL
LIN {X 0,Y 601.431,Z 701.561,A -85,B 0,C 180,E1 -731.012,E2 -731.012} C_VEL
LIN {X 0,Y 601.407,Z 701.567,A -85,B 0,C 180,E1 -733.516,E2 -733.516} C_VEL
LIN {X 0,Y 601.443,Z 701.568,A -85,B 0,C 180,E1 -736.287,E2 -736.287} C_VEL
LIN {X 0,Y 601.419,Z 701.563,A -85,B 0,C 180,E1 -739.099,E2 -739.099} C_VEL
LIN {X 0,Y 601.406,Z 701.564,A -85,B 0,C 180,E1 -741.239,E2 -741.239} C_VEL
LIN {X 0,Y 601.454,Z 701.567,A -85,B 0,C 180,E1 -744.141,E2 -744.141} C_VEL
LIN {X 0,Y 601.455,Z 701.559,A -85,B 0,C 180,E1 -747.111,E2 -747.111} C_VEL
LIN {X 0,Y 601.417,Z 701.563,A -85,B 0,C 180,E1 -749.393,E2 -749.393} C_VEL
LIN {X 0,Y 601.405,Z 701.566,A -85,B 0,C 180,E1 -751.727,E2 -751.727} C_VEL
LIN {X 0,Y 601.433,Z 701.566,A -85,B 0,C 180,E1 -754.118,E2 -754.118} C_VEL
LIN {X 0,Y 601.439,Z 701.561,A -85,B 0,C 180,E1 -757.382,E2 -757.382} C_VEL
LIN {X 0,Y 601.414,Z 701.566,A -85,B 0,C 180,E1 -759.995,E2 -759.995} C_VEL
LIN {X 0,Y 601.415,Z 701.574,A -85,B 0,C 180,E1 -762.67,E2 -762.67} C_VEL
LIN {X 0,Y 601.43,Z 701.562,A -85,B 0,C 180,E1 -765.482,E2 -765.482} C_VEL
LIN {X 0,Y 601.429,Z 701.568,A -85,B 0,C 180,E1 -768.407,E2 -768.407} C_VEL
LIN {X 0,Y 601.437,Z 701.563,A -85,B 0,C 180,E1 -771.529,E2 -771.529} C_VEL
LIN {X 0,Y 601.437,Z 701.591,A -85,B 0,C 180,E1 -773.888,E2 -773.888} C_VEL
LIN {X 0,Y 601.868,Z 705.249,A -85,B 0,C 180,E1 -774.602,E2 -774.602} C_VEL
LIN {X 0,Y 601.79,Z 718.14,A -85,B 0,C 180,E1 -777.23,E2 -777.23} C_VEL
LIN {X 0,Y 601.728,Z 731.234,A -85,B 0,C 180,E1 -779.852,E2 -779.852} C_VEL
LIN {X 0,Y 601.67,Z 745.284,A -85,B 0,C 180,E1 -782.591,E2 -782.591} C_VEL
LIN {X 0,Y 601.593,Z 758.624,A -85,B 0,C 180,E1 -785.13,E2 -785.13} C_VEL
LIN {X 0,Y 601.54,Z 772.418,A -85,B 0,C 180,E1 -787.703,E2 -787.703} C_VEL
LIN {X 0,Y 601.514,Z 786.014,A -85,B 0,C 180,E1 -790.194,E2 -790.194} C_VEL
LIN {X 0,Y 601.44,Z 801.665,A -85,B 0,C 180,E1 -793.014,E2 -793.014} C_VEL
LIN {X 0,Y 601.431,Z 815.36,A -85,B 0,C 180,E1 -795.449,E2 -795.449} C_VEL
LIN {X 0,Y 601.408,Z 830.156,A -85,B 0,C 180,E1 -798.05,E2 -798.05} C_VEL
LIN {X 0,Y 601.594,Z 843.347,A -85,B 0,C 180,E1 -798.289,E2 -798.289} C_VEL
LIN {X 0,Y 601.562,Z 856.436,A -85,B 0,C 180,E1 -798.662,E2 -798.662} C_VEL
LIN {X 0,Y 601.511,Z 868.678,A -85,B 0,C 180,E1 -799.153,E2 -799.153} C_VEL
LIN {X 0,Y 601.479,Z 879.754,A -85,B 0,C 180,E1 -799.736,E2 -799.736} C_VEL
LIN {X 0,Y 601.462,Z 891.251,A -85,B 0,C 180,E1 -800.5,E2 -800.5} C_VEL
LIN {X 0,Y 601.436,Z 900.535,A -85,B 0,C 180,E1 -801.262,E2 -801.262} C_VEL
LIN {X 0,Y 601.4,Z 908.988,A -85,B 0,C 180,E1 -802.108,E2 -802.108} C_VEL
LIN {X 0,Y 601.382,Z 917.234,A -85,B 0,C 180,E1 -803.12,E2 -803.12} C_VEL
LIN {X 0,Y 601.372,Z 923.876,A -85,B 0,C 180,E1 -804.131,E2 -804.131} C_VEL
LIN {X 0,Y 601.336,Z 929.95,A -85,B 0,C 180,E1 -805.307,E2 -805.307} C_VEL
LIN {X 0,Y 601.367,Z 933.896,A -85,B 0,C 180,E1 -806.315,E2 -806.315} C_VEL
LIN {X 0,Y 601.325,Z 936.809,A -85,B 0,C 180,E1 -807.32,E2 -807.32} C_VEL
LIN {X 0,Y 601.34,Z 938.201,A -85,B 0,C 180,E1 -807.991,E2 -807.991} C_VEL
LIN {X 0,Y 601.339,Z 939.784,A -85,B 0,C 180,E1 -809.33,E2 -809.33} C_VEL
LIN {X 0,Y 601.335,Z 940,A -85,B 0,C 180,E1 -810,E2 -810} C_VEL
LIN {X 0,Y 601.348,Z 939.184,A -85,B 0,C 180,E1 -811.339,E2 -811.339} C_VEL
LIN {X 0,Y 601.34,Z 938.202,A -85,B 0,C 180,E1 -812.009,E2 -812.009} C_VEL
LIN {X 0,Y 601.325,Z 936.809,A -85,B 0,C 180,E1 -812.68,E2 -812.68} C_VEL
LIN {X 0,Y 601.367,Z 933.896,A -85,B 0,C 180,E1 -813.685,E2 -813.685} C_VEL
LIN {X 0,Y 601.336,Z 929.95,A -85,B 0,C 180,E1 -814.693,E2 -814.693} C_VEL
LIN {X 0,Y 601.372,Z 923.877,A -85,B 0,C 180,E1 -815.869,E2 -815.869} C_VEL
LIN {X 0,Y 601.382,Z 917.235,A -85,B 0,C 180,E1 -816.88,E2 -816.88} C_VEL
LIN {X 0,Y 601.4,Z 908.989,A -85,B 0,C 180,E1 -817.892,E2 -817.892} C_VEL
LIN {X 0,Y 601.436,Z 900.537,A -85,B 0,C 180,E1 -818.738,E2 -818.738} C_VEL
LIN {X 0,Y 601.446,Z 890.092,A -85,B 0,C 180,E1 -819.585,E2 -819.585} C_VEL
LIN {X 0,Y 601.479,Z 879.757,A -85,B 0,C 180,E1 -820.264,E2 -820.264} C_VEL
LIN {X 0,Y 601.508,Z 867.937,A -85,B 0,C 180,E1 -820.882,E2 -820.882} C_VEL
LIN {X 0,Y 601.566,Z 855.28,A -85,B 0,C 180,E1 -821.376,E2 -821.376} C_VEL
LIN {X 0,Y 601.585,Z 842.438,A -85,B 0,C 180,E1 -821.733,E2 -821.733} C_VEL
LIN {X 0,Y 601.408,Z 830.157,A -85,B 0,C 180,E1 -821.95,E2 -821.95} C_VEL
LIN {X 0,Y 601.431,Z 815.361,A -85,B 0,C 180,E1 -824.551,E2 -824.551} C_VEL
LIN {X 0,Y 601.47,Z 799.71,A -85,B 0,C 180,E1 -827.335,E2 -827.335} C_VEL
LIN {X 0,Y 601.51,Z 784.058,A -85,B 0,C 180,E1 -830.162,E2 -830.162} C_VEL
LIN {X 0,Y 601.577,Z 768.407,A -85,B 0,C 180,E1 -833.04,E2 -833.04} C_VEL
LIN {X 0,Y 601.642,Z 753.112,A -85,B 0,C 180,E1 -835.912,E2 -835.912} C_VEL
LIN {X 0,Y 601.69,Z 739.06,A -85,B 0,C 180,E1 -838.614,E2 -838.614} C_VEL
LIN {X 0,Y 601.745,Z 725.864,A -85,B 0,C 180,E1 -841.214,E2 -841.214} C_VEL
LIN {X 0,Y 601.861,Z 712.129,A -85,B 0,C 180,E1 -843.996,E2 -843.996} C_VEL
LIN {X 0,Y 601.813,Z 703.604,A -85,B 0,C 180,E1 -845.726,E2 -845.726} C_VEL
LIN {X 0,Y 601.442,Z 701.565,A -85,B 0,C 180,E1 -846.158,E2 -846.158} C_VEL
LIN {X 0,Y 601.437,Z 701.571,A -85,B 0,C 180,E1 -849.125,E2 -849.125} C_VEL
LIN {X 0,Y 601.43,Z 701.565,A -85,B 0,C 180,E1 -851.765,E2 -851.765} C_VEL
LIN {X 0,Y 601.428,Z 701.563,A -85,B 0,C 180,E1 -854.535,E2 -854.535} C_VEL
LIN {X 0,Y 601.413,Z 701.575,A -85,B 0,C 180,E1 -857.409,E2 -857.409} C_VEL
LIN {X 0,Y 601.442,Z 701.56,A -85,B 0,C 180,E1 -860.464,E2 -860.464} C_VEL
LIN {X 0,Y 601.404,Z 701.575,A -85,B 0,C 180,E1 -863.417,E2 -863.417} C_VEL
LIN {X 0,Y 601.435,Z 701.563,A -85,B 0,C 180,E1 -866.064,E2 -866.064} C_VEL
LIN {X 0,Y 601.423,Z 701.562,A -85,B 0,C 180,E1 -868.545,E2 -868.545} C_VEL
LIN {X 0,Y 601.438,Z 701.567,A -85,B 0,C 180,E1 -871.373,E2 -871.373} C_VEL
LIN {X 0,Y 601.404,Z 701.576,A -85,B 0,C 180,E1 -873.636,E2 -873.636} C_VEL
LIN {X 0,Y 601.453,Z 701.567,A -85,B 0,C 180,E1 -875.859,E2 -875.859} C_VEL
LIN {X 0,Y 601.405,Z 701.565,A -85,B 0,C 180,E1 -878.761,E2 -878.761} C_VEL
LIN {X 0,Y 601.422,Z 701.57,A -85,B 0,C 180,E1 -881.608,E2 -881.608} C_VEL
LIN {X 0,Y 601.441,Z 701.569,A -85,B 0,C 180,E1 -883.713,E2 -883.713} C_VEL
LIN {X 0,Y 601.404,Z 701.567,A -85,B 0,C 180,E1 -886.484,E2 -886.484} C_VEL
LIN {X 0,Y 601.422,Z 701.564,A -85,B 0,C 180,E1 -889.224,E2 -889.224} C_VEL
LIN {X 0,Y 601.442,Z 701.571,A -85,B 0,C 180,E1 -891.939,E2 -891.939} C_VEL
LIN {X 0,Y 601.409,Z 701.566,A -85,B 0,C 180,E1 -894.636,E2 -894.636} C_VEL
LIN {X 0,Y 601.444,Z 701.561,A -85,B 0,C 180,E1 -897.321,E2 -897.321} C_VEL
LIN {X 0,Y 601.452,Z 701.568,A -85,B 0,C 180,E1 -900,E2 -900} C_VEL
LIN {X 0,Y 601.42,Z 701.566,A -85,B 0,C 180,E1 -902.679,E2 -902.679} C_VEL
LIN {X 0,Y 601.411,Z 701.564,A -85,B 0,C 180,E1 -905.364,E2 -905.364} C_VEL
LIN {X 0,Y 601.443,Z 701.568,A -85,B 0,C 180,E1 -908.061,E2 -908.061} C_VEL
LIN {X 0,Y 601.397,Z 701.567,A -85,B 0,C 180,E1 -910.997,E2 -910.997} C_VEL
LIN {X 0,Y 601.402,Z 701.57,A -85,B 0,C 180,E1 -912.354,E2 -912.354} C_VEL
LIN {X 0,Y 600.724,Z 701.653,A -85,B 0,C 180,E1 -912.913,E2 -912.913} C_VEL
LIN {X 0,Y 597.866,Z 702.008,A -85,B 0,C 180,E1 -913.821,E2 -913.821} C_VEL
LIN {X 0,Y 595.457,Z 702.314,A -85,B 0,C 180,E1 -914.551,E2 -914.551} C_VEL
LIN {X 0,Y 594.423,Z 702.436,A -85,B 0,C 180,E1 -915.115,E2 -915.115} C_VEL
LIN {X 0,Y 594.339,Z 702.445,A -85,B 0,C 180,E1 -915.306,E2 -915.306} C_VEL
LIN {X 0,Y 594.342,Z 702.447,A -85,B 0,C 180,E1 -917.906,E2 -917.906} C_VEL
LIN {X 0,Y 594.401,Z 702.443,A -85,B 0,C 180,E1 -920.776,E2 -920.776} C_VEL
LIN {X 0,Y 594.365,Z 702.442,A -85,B 0,C 180,E1 -923.705,E2 -923.705} C_VEL
LIN {X 0,Y 594.351,Z 702.453,A -85,B 0,C 180,E1 -926.701,E2 -926.701} C_VEL
LIN {X 0,Y 594.375,Z 702.445,A -85,B 0,C 180,E1 -928.999,E2 -928.999} C_VEL
LIN {X 0,Y 594.368,Z 702.442,A -85,B 0,C 180,E1 -931.641,E2 -931.641} C_VEL
LIN {X 0,Y 594.375,Z 702.449,A -85,B 0,C 180,E1 -934.581,E2 -934.581} C_VEL
LIN {X 0,Y 594.353,Z 702.444,A -85,B 0,C 180,E1 -937.603,E2 -937.603} C_VEL
LIN {X 0,Y 594.332,Z 702.446,A -85,B 0,C 180,E1 -939.769,E2 -939.769} C_VEL
LIN {X 0,Y 594.341,Z 702.448,A -85,B 0,C 180,E1 -942.378,E2 -942.378} C_VEL
LIN {X 0,Y 594.34,Z 702.451,A -85,B 0,C 180,E1 -945.194,E2 -945.194} C_VEL
LIN {X 0,Y 594.356,Z 702.443,A -85,B 0,C 180,E1 -948.155,E2 -948.155} C_VEL
LIN {X 0,Y 594.364,Z 702.448,A -85,B 0,C 180,E1 -951.299,E2 -951.299} C_VEL
LIN {X 0,Y 594.327,Z 702.448,A -85,B 0,C 180,E1 -953.754,E2 -953.754} C_VEL
LIN {X 0,Y 594.32,Z 702.448,A -85,B 0,C 180,E1 -956.235,E2 -956.235} C_VEL
LIN {X 0,Y 594.34,Z 702.448,A -85,B 0,C 180,E1 -958.648,E2 -958.648} C_VEL
LIN {X 0,Y 594.377,Z 702.449,A -85,B 0,C 180,E1 -961.044,E2 -961.044} C_VEL
LIN {X 0,Y 594.323,Z 702.448,A -85,B 0,C 180,E1 -964.053,E2 -964.053} C_VEL
LIN {X 0,Y 594.344,Z 702.445,A -85,B 0,C 180,E1 -966.294,E2 -966.294} C_VEL
LIN {X 0,Y 594.405,Z 702.446,A -85,B 0,C 180,E1 -969.224,E2 -969.224} C_VEL
LIN {X 0,Y 594.319,Z 702.448,A -85,B 0,C 180,E1 -972.094,E2 -972.094} C_VEL
LIN {X 0,Y 594.331,Z 702.447,A -85,B 0,C 180,E1 -974.218,E2 -974.218} C_VEL
LIN {X 0,Y 594.34,Z 702.448,A -85,B 0,C 180,E1 -977.016,E2 -977.016} C_VEL
LIN {X 0,Y 594.337,Z 702.452,A -85,B 0,C 180,E1 -979.783,E2 -979.783} C_VEL
LIN {X 0,Y 594.34,Z 702.445,A -85,B 0,C 180,E1 -982.526,E2 -982.526} C_VEL
LIN {X 0,Y 594.368,Z 702.446,A -85,B 0,C 180,E1 -985.252,E2 -985.252} C_VEL
LIN {X 0,Y 594.395,Z 702.444,A -85,B 0,C 180,E1 -987.967,E2 -987.967} C_VEL
LIN {X 0,Y 594.414,Z 702.441,A -85,B 0,C 180,E1 -990,E2 -990} C_VEL
LIN {X 0,Y 594.371,Z 702.441,A -85,B 0,C 180,E1 -992.711,E2 -992.711} C_VEL
LIN {X 0,Y 594.368,Z 702.446,A -85,B 0,C 180,E1 -995.428,E2 -995.428} C_VEL
LIN {X 0,Y 594.381,Z 702.445,A -85,B 0,C 180,E1 -998.157,E2 -998.157} C_VEL
LIN {X 0,Y 594.368,Z 702.442,A -85,B 0,C 180,E1 -1001.061,E2 -1001.061} C_VEL
LIN {X 0,Y 594.371,Z 702.448,A -85,B 0,C 180,E1 -1003.679,E2 -1003.679} C_VEL
LIN {X 0,Y 594.365,Z 702.443,A -85,B 0,C 180,E1 -1006.708,E2 -1006.708} C_VEL
LIN {X 0,Y 594.362,Z 702.443,A -85,B 0,C 180,E1 -1009.335,E2 -1009.335} C_VEL
LIN {X 0,Y 594.359,Z 702.445,A -85,B 0,C 180,E1 -1011.504,E2 -1011.504} C_VEL
LIN {X 0,Y 594.393,Z 702.443,A -85,B 0,C 180,E1 -1014.446,E2 -1014.446} C_VEL
LIN {X 0,Y 594.36,Z 702.445,A -85,B 0,C 180,E1 -1016.701,E2 -1016.701} C_VEL
LIN {X 0,Y 594.383,Z 702.44,A -85,B 0,C 180,E1 -1018.999,E2 -1018.999} C_VEL
LIN {X 0,Y 594.376,Z 702.442,A -85,B 0,C 180,E1 -1021.642,E2 -1021.642} C_VEL
LIN {X 0,Y 594.381,Z 702.446,A -85,B 0,C 180,E1 -1024.58,E2 -1024.58} C_VEL
LIN {X 0,Y 594.39,Z 702.439,A -85,B 0,C 180,E1 -1027.608,E2 -1027.608} C_VEL
LIN {X 0,Y 594.368,Z 702.449,A -85,B 0,C 180,E1 -1030.567,E2 -1030.567} C_VEL
LIN {X 0,Y 594.371,Z 702.441,A -85,B 0,C 180,E1 -1033.299,E2 -1033.299} C_VEL
LIN {X 0,Y 594.364,Z 702.447,A -85,B 0,C 180,E1 -1036.161,E2 -1036.161} C_VEL
LIN {X 0,Y 594.382,Z 702.451,A -85,B 0,C 180,E1 -1038.536,E2 -1038.536} C_VEL
LIN {X 0,Y 594.4,Z 702.447,A -85,B 0,C 180,E1 -1040.431,E2 -1040.431} C_VEL
LIN {X 0,Y 594.566,Z 714.435,A -85,B 0,C 180,E1 -1040.882,E2 -1040.882} C_VEL
LIN {X 0,Y 594.519,Z 726.575,A -85,B 0,C 180,E1 -1041.476,E2 -1041.476} C_VEL
LIN {X 0,Y 594.437,Z 737.536,A -85,B 0,C 180,E1 -1042.159,E2 -1042.159} C_VEL
LIN {X 0,Y 594.395,Z 747.257,A -85,B 0,C 180,E1 -1042.914,E2 -1042.914} C_VEL
LIN {X 0,Y 594.358,Z 756.152,A -85,B 0,C 180,E1 -1043.756,E2 -1043.756} C_VEL
LIN {X 0,Y 594.344,Z 764.173,A -85,B 0,C 180,E1 -1044.678,E2 -1044.678} C_VEL
LIN {X 0,Y 594.289,Z 771.216,A -85,B 0,C 180,E1 -1045.67,E2 -1045.67} C_VEL
LIN {X 0,Y 594.276,Z 776.781,A -85,B 0,C 180,E1 -1046.638,E2 -1046.638} C_VEL
LIN {X 0,Y 594.255,Z 782.209,A -85,B 0,C 180,E1 -1047.846,E2 -1047.846} C_VEL
LIN {X 0,Y 594.241,Z 786.044,A -85,B 0,C 180,E1 -1049.038,E2 -1049.038} C_VEL
LIN {X 0,Y 594.234,Z 788.534,A -85,B 0,C 180,E1 -1050.216,E2 -1050.216} C_VEL
LIN {X 0,Y 594.254,Z 789.577,A -85,B 0,C 180,E1 -1051.065,E2 -1051.065} C_VEL
LIN {X 0,Y 594.221,Z 789.942,A -85,B 0,C 180,E1 -1051.765,E2 -1051.765} C_VEL
LIN {X 0,Y 594.266,Z 789.877,A -85,B 0,C 180,E1 -1052.533,E2 -1052.533} C_VEL
LIN {X 0,Y 594.225,Z 789.307,A -85,B 0,C 180,E1 -1053.293,E2 -1053.293} C_VEL
LIN {X 0,Y 594.229,Z 788.251,A -85,B 0,C 180,E1 -1054.049,E2 -1054.049} C_VEL
LIN {X 0,Y 594.25,Z 785.723,A -85,B 0,C 180,E1 -1055.175,E2 -1055.175} C_VEL
LIN {X 0,Y 594.251,Z 782.036,A -85,B 0,C 180,E1 -1056.29,E2 -1056.29} C_VEL
LIN {X 0,Y 594.276,Z 776.391,A -85,B 0,C 180,E1 -1057.525,E2 -1057.525} C_VEL
LIN {X 0,Y 594.305,Z 770.734,A -85,B 0,C 180,E1 -1058.494,E2 -1058.494} C_VEL
LIN {X 0,Y 594.32,Z 762.813,A -85,B 0,C 180,E1 -1059.583,E2 -1059.583} C_VEL
LIN {X 0,Y 594.375,Z 754.706,A -85,B 0,C 180,E1 -1060.486,E2 -1060.486} C_VEL
LIN {X 0,Y 594.413,Z 744.761,A -85,B 0,C 180,E1 -1061.383,E2 -1061.383} C_VEL
LIN {X 0,Y 594.472,Z 733.676,A -85,B 0,C 180,E1 -1062.187,E2 -1062.187} C_VEL
LIN {X 0,Y 594.478,Z 722.949,A -85,B 0,C 180,E1 -1062.809,E2 -1062.809} C_VEL
LIN {X 0,Y 594.567,Z 710.748,A -85,B 0,C 180,E1 -1063.359,E2 -1063.359} C_VEL
LIN {X 0,Y 594.422,Z 702.444,A -85,B 0,C 180,E1 -1063.67,E2 -1063.67} C_VEL
LIN {X 0,Y 594.374,Z 702.442,A -85,B 0,C 180,E1 -1066.321,E2 -1066.321} C_VEL
LIN {X 0,Y 594.353,Z 702.447,A -85,B 0,C 180,E1 -1069.094,E2 -1069.094} C_VEL
LIN {X 0,Y 594.415,Z 702.443,A -85,B 0,C 180,E1 -1071.843,E2 -1071.843} C_VEL
LIN {X 0,Y 594.38,Z 702.44,A -85,B 0,C 180,E1 -1074.572,E2 -1074.572} C_VEL
LIN {X 0,Y 594.393,Z 702.442,A -85,B 0,C 180,E1 -1077.289,E2 -1077.289} C_VEL
LIN {X 0,Y 594.421,Z 702.443,A -85,B 0,C 180,E1 -1080,E2 -1080} C_VEL
LIN {X 0,Y 594.411,Z 702.436,A -85,B 0,C 180,E1 -1082.711,E2 -1082.711} C_VEL
LIN {X 0,Y 594.38,Z 702.443,A -85,B 0,C 180,E1 -1085.428,E2 -1085.428} C_VEL
LIN {X 0,Y 594.387,Z 702.446,A -85,B 0,C 180,E1 -1088.157,E2 -1088.157} C_VEL
LIN {X 0,Y 594.395,Z 702.438,A -85,B 0,C 180,E1 -1091.074,E2 -1091.074} C_VEL
LIN {X 0,Y 594.377,Z 702.444,A -85,B 0,C 180,E1 -1093.679,E2 -1093.679} C_VEL
LIN {X 0,Y 594.4,Z 702.439,A -85,B 0,C 180,E1 -1096.719,E2 -1096.719} C_VEL
LIN {X 0,Y 594.369,Z 702.441,A -85,B 0,C 180,E1 -1099.334,E2 -1099.334} C_VEL
LIN {X 0,Y 594.367,Z 702.442,A -85,B 0,C 180,E1 -1101.503,E2 -1101.503} C_VEL
LIN {X 0,Y 594.393,Z 702.446,A -85,B 0,C 180,E1 -1104.446,E2 -1104.446} C_VEL
LIN {X 0,Y 594.387,Z 702.443,A -85,B 0,C 180,E1 -1106.699,E2 -1106.699} C_VEL
LIN {X 0,Y 594.385,Z 702.441,A -85,B 0,C 180,E1 -1108.998,E2 -1108.998} C_VEL
LIN {X 0,Y 594.381,Z 702.44,A -85,B 0,C 180,E1 -1111.643,E2 -1111.643} C_VEL
LIN {X 0,Y 594.4,Z 702.447,A -85,B 0,C 180,E1 -1114.579,E2 -1114.579} C_VEL
LIN {X 0,Y 594.392,Z 702.439,A -85,B 0,C 180,E1 -1117.608,E2 -1117.608} C_VEL
LIN {X 0,Y 594.372,Z 702.452,A -85,B 0,C 180,E1 -1120.567,E2 -1120.567} C_VEL
LIN {X 0,Y 594.37,Z 702.443,A -85,B 0,C 180,E1 -1123.299,E2 -1123.299} C_VEL
LIN {X 0,Y 594.372,Z 702.444,A -85,B 0,C 180,E1 -1126.16,E2 -1126.16} C_VEL
LIN {X 0,Y 594.386,Z 702.448,A -85,B 0,C 180,E1 -1128.536,E2 -1128.536} C_VEL
LIN {X 0,Y 594.387,Z 702.444,A -85,B 0,C 180,E1 -1131.296,E2 -1131.296} C_VEL
LIN {X 0,Y 594.413,Z 702.503,A -85,B 0,C 180,E1 -1133.729,E2 -1133.729} C_VEL
LIN {X 0,Y 594.955,Z 706.931,A -85,B 0,C 180,E1 -1134.595,E2 -1134.595} C_VEL
LIN {X 0,Y 594.987,Z 715.582,A -85,B 0,C 180,E1 -1136.278,E2 -1136.278} C_VEL
LIN {X 0,Y 594.896,Z 727.321,A -85,B 0,C 180,E1 -1138.68,E2 -1138.68} C_VEL
LIN {X 0,Y 594.787,Z 741.016,A -85,B 0,C 180,E1 -1141.409,E2 -1141.409} C_VEL
LIN {X 0,Y 594.699,Z 756.667,A -85,B 0,C 180,E1 -1144.447,E2 -1144.447} C_VEL
LIN {X 0,Y 594.632,Z 771.218,A -85,B 0,C 180,E1 -1147.204,E2 -1147.204} C_VEL
LIN {X 0,Y 594.532,Z 786.014,A -85,B 0,C 180,E1 -1149.952,E2 -1149.952} C_VEL
LIN {X 0,Y 594.459,Z 799.709,A -85,B 0,C 180,E1 -1152.454,E2 -1152.454} C_VEL
LIN {X 0,Y 594.392,Z 815.36,A -85,B 0,C 180,E1 -1155.273,E2 -1155.273} C_VEL
LIN {X 0,Y 594.354,Z 830.156,A -85,B 0,C 180,E1 -1157.906,E2 -1157.906} C_VEL
LIN {X 0,Y 594.67,Z 835.939,A -85,B 0,C 180,E1 -1157.999,E2 -1157.999} C_VEL
LIN {X 0,Y 594.652,Z 849.212,A -85,B 0,C 180,E1 -1158.301,E2 -1158.301} C_VEL
LIN {X 0,Y 594.562,Z 862.297,A -85,B 0,C 180,E1 -1158.746,E2 -1158.746} C_VEL
LIN {X 0,Y 594.518,Z 873.631,A -85,B 0,C 180,E1 -1159.27,E2 -1159.27} C_VEL
LIN {X 0,Y 594.468,Z 885.197,A -85,B 0,C 180,E1 -1159.957,E2 -1159.957} C_VEL
LIN {X 0,Y 594.414,Z 895.594,A -85,B 0,C 180,E1 -1160.729,E2 -1160.729} C_VEL
LIN {X 0,Y 594.383,Z 904.111,A -85,B 0,C 180,E1 -1161.5,E2 -1161.5} C_VEL
LIN {X 0,Y 594.347,Z 911.959,A -85,B 0,C 180,E1 -1162.355,E2 -1162.355} C_VEL
LIN {X 0,Y 594.283,Z 919.812,A -85,B 0,C 180,E1 -1163.408,E2 -1163.408} C_VEL
LIN {X 0,Y 594.289,Z 926.68,A -85,B 0,C 180,E1 -1164.571,E2 -1164.571} C_VEL
LIN {X 0,Y 594.27,Z 931.371,A -85,B 0,C 180,E1 -1165.591,E2 -1165.591} C_VEL
LIN {X 0,Y 594.268,Z 934.956,A -85,B 0,C 180,E1 -1166.61,E2 -1166.61} C_VEL
LIN {X 0,Y 594.226,Z 936.809,A -85,B 0,C 180,E1 -1167.288,E2 -1167.288} C_VEL
LIN {X 0,Y 594.239,Z 938.202,A -85,B 0,C 180,E1 -1167.967,E2 -1167.967} C_VEL
LIN {X 0,Y 594.239,Z 939.784,A -85,B 0,C 180,E1 -1169.322,E2 -1169.322} C_VEL
LIN {X 0,Y 594.236,Z 940,A -85,B 0,C 180,E1 -1170,E2 -1170} C_VEL
LIN {X 0,Y 594.247,Z 939.185,A -85,B 0,C 180,E1 -1171.355,E2 -1171.355} C_VEL
LIN {X 0,Y 594.239,Z 938.202,A -85,B 0,C 180,E1 -1172.033,E2 -1172.033} C_VEL
LIN {X 0,Y 594.226,Z 936.81,A -85,B 0,C 180,E1 -1172.712,E2 -1172.712} C_VEL
LIN {X 0,Y 594.289,Z 933.896,A -85,B 0,C 180,E1 -1173.729,E2 -1173.729} C_VEL
LIN {X 0,Y 594.241,Z 929.95,A -85,B 0,C 180,E1 -1174.749,E2 -1174.749} C_VEL
LIN {X 0,Y 594.304,Z 923.877,A -85,B 0,C 180,E1 -1175.939,E2 -1175.939} C_VEL
LIN {X 0,Y 594.308,Z 917.236,A -85,B 0,C 180,E1 -1176.962,E2 -1176.962} C_VEL
LIN {X 0,Y 594.359,Z 908.99,A -85,B 0,C 180,E1 -1177.986,E2 -1177.986} C_VEL
LIN {X 0,Y 594.382,Z 900.537,A -85,B 0,C 180,E1 -1178.842,E2 -1178.842} C_VEL
LIN {X 0,Y 594.429,Z 890.093,A -85,B 0,C 180,E1 -1179.699,E2 -1179.699} C_VEL
LIN {X 0,Y 594.487,Z 879.758,A -85,B 0,C 180,E1 -1180.386,E2 -1180.386} C_VEL
LIN {X 0,Y 594.524,Z 868.848,A -85,B 0,C 180,E1 -1180.968,E2 -1180.968} C_VEL
LIN {X 0,Y 594.597,Z 856.748,A -85,B 0,C 180,E1 -1181.463,E2 -1181.463} C_VEL
LIN {X 0,Y 594.651,Z 843.352,A -85,B 0,C 180,E1 -1181.85,E2 -1181.85} C_VEL
LIN {X 0,Y 594.56,Z 831.601,A -85,B 0,C 180,E1 -1182.068,E2 -1182.068} C_VEL
LIN {X 0,Y 594.359,Z 830.034,A -85,B 0,C 180,E1 -1182.116,E2 -1182.116} C_VEL
LIN {X 0,Y 594.392,Z 815.361,A -85,B 0,C 180,E1 -1184.727,E2 -1184.727} C_VEL
LIN {X 0,Y 594.464,Z 799.71,A -85,B 0,C 180,E1 -1187.546,E2 -1187.546} C_VEL
LIN {X 0,Y 594.53,Z 784.058,A -85,B 0,C 180,E1 -1190.409,E2 -1190.409} C_VEL
LIN {X 0,Y 594.617,Z 770.363,A -85,B 0,C 180,E1 -1192.957,E2 -1192.957} C_VEL
LIN {X 0,Y 594.706,Z 754.712,A -85,B 0,C 180,E1 -1195.929,E2 -1195.929} C_VEL
LIN {X 0,Y 594.787,Z 741.017,A -85,B 0,C 180,E1 -1198.591,E2 -1198.591} C_VEL
LIN {X 0,Y 594.895,Z 727.322,A -85,B 0,C 180,E1 -1201.32,E2 -1201.32} C_VEL
LIN {X 0,Y 595.013,Z 714.361,A -85,B 0,C 180,E1 -1203.975,E2 -1203.975} C_VEL
LIN {X 0,Y 594.927,Z 705.22,A -85,B 0,C 180,E1 -1205.785,E2 -1205.785} C_VEL
LIN {X 0,Y 594.408,Z 702.443,A -85,B 0,C 180,E1 -1206.424,E2 -1206.424} C_VEL
LIN {X 0,Y 594.39,Z 702.445,A -85,B 0,C 180,E1 -1208.805,E2 -1208.805} C_VEL
LIN {X 0,Y 594.388,Z 702.441,A -85,B 0,C 180,E1 -1211.849,E2 -1211.849} C_VEL
LIN {X 0,Y 594.367,Z 702.444,A -85,B 0,C 180,E1 -1214.809,E2 -1214.809} C_VEL
LIN {X 0,Y 594.37,Z 702.448,A -85,B 0,C 180,E1 -1217.625,E2 -1217.625} C_VEL
LIN {X 0,Y 594.394,Z 702.438,A -85,B 0,C 180,E1 -1220.321,E2 -1220.321} C_VEL
LIN {X 0,Y 594.385,Z 702.441,A -85,B 0,C 180,E1 -1222.913,E2 -1222.913} C_VEL
LIN {X 0,Y 594.386,Z 702.444,A -85,B 0,C 180,E1 -1225.861,E2 -1225.861} C_VEL
LIN {X 0,Y 594.373,Z 702.441,A -85,B 0,C 180,E1 -1228.65,E2 -1228.65} C_VEL
LIN {X 0,Y 594.387,Z 702.441,A -85,B 0,C 180,E1 -1231.042,E2 -1231.042} C_VEL
LIN {X 0,Y 594.388,Z 702.444,A -85,B 0,C 180,E1 -1233.301,E2 -1233.301} C_VEL
LIN {X 0,Y 594.375,Z 702.442,A -85,B 0,C 180,E1 -1236.295,E2 -1236.295} C_VEL
LIN {X 0,Y 594.409,Z 702.439,A -85,B 0,C 180,E1 -1239.225,E2 -1239.225} C_VEL
LIN {X 0,Y 594.351,Z 702.449,A -85,B 0,C 180,E1 -1242.095,E2 -1242.095} C_VEL
LIN {X 0,Y 594.362,Z 702.447,A -85,B 0,C 180,E1 -1244.219,E2 -1244.219} C_VEL
LIN {X 0,Y 594.374,Z 702.444,A -85,B 0,C 180,E1 -1246.321,E2 -1246.321} C_VEL
LIN {X 0,Y 594.38,Z 702.44,A -85,B 0,C 180,E1 -1249.095,E2 -1249.095} C_VEL
LIN {X 0,Y 594.415,Z 702.444,A -85,B 0,C 180,E1 -1251.843,E2 -1251.843} C_VEL
LIN {X 0,Y 594.376,Z 702.443,A -85,B 0,C 180,E1 -1254.572,E2 -1254.572} C_VEL
LIN {X 0,Y 594.407,Z 702.437,A -85,B 0,C 180,E1 -1257.289,E2 -1257.289} C_VEL
LIN {X 0,Y 594.42,Z 702.444,A -85,B 0,C 180,E1 -1260,E2 -1260} C_VEL
LIN {X 0,Y 594.389,Z 702.441,A -85,B 0,C 180,E1 -1262.711,E2 -1262.711} C_VEL
LIN {X 0,Y 594.378,Z 702.441,A -85,B 0,C 180,E1 -1265.428,E2 -1265.428} C_VEL
LIN {X 0,Y 594.414,Z 702.445,A -85,B 0,C 180,E1 -1268.157,E2 -1268.157} C_VEL
LIN {X 0,Y 594.367,Z 702.442,A -85,B 0,C 180,E1 -1271.061,E2 -1271.061} C_VEL
LIN {X 0,Y 594.371,Z 702.442,A -85,B 0,C 180,E1 -1273.679,E2 -1273.679} C_VEL
LIN {X 0,Y 594.339,Z 702.445,A -85,B 0,C 180,E1 -1275.306,E2 -1275.306} C_VEL
LIN {X 0,Y 593.67,Z 702.532,A -85,B 0,C 180,E1 -1275.871,E2 -1275.871} C_VEL
LIN {X 0,Y 590.809,Z 702.89,A -85,B 0,C 180,E1 -1276.789,E2 -1276.789} C_VEL
LIN {X 0,Y 588.4,Z 703.191,A -85,B 0,C 180,E1 -1277.528,E2 -1277.528} C_VEL
LIN {X 0,Y 587.376,Z 703.318,A -85,B 0,C 180,E1 -1278.098,E2 -1278.098} C_VEL
LIN {X 0,Y 587.298,Z 703.327,A -85,B 0,C 180,E1 -1278.291,E2 -1278.291} C_VEL
LIN {X 0,Y 587.335,Z 703.32,A -85,B 0,C 180,E1 -1281.038,E2 -1281.038} C_VEL
LIN {X 0,Y 587.308,Z 703.322,A -85,B 0,C 180,E1 -1283.26,E2 -1283.26} C_VEL
LIN {X 0,Y 587.295,Z 703.323,A -85,B 0,C 180,E1 -1285.519,E2 -1285.519} C_VEL
LIN {X 0,Y 587.303,Z 703.322,A -85,B 0,C 180,E1 -1287.82,E2 -1287.82} C_VEL
LIN {X 0,Y 587.32,Z 703.328,A -85,B 0,C 180,E1 -1290.507,E2 -1290.507} C_VEL
LIN {X 0,Y 587.335,Z 703.322,A -85,B 0,C 180,E1 -1293.111,E2 -1293.111} C_VEL
LIN {X 0,Y 587.28,Z 703.325,A -85,B 0,C 180,E1 -1295.901,E2 -1295.901} C_VEL
LIN {X 0,Y 587.311,Z 703.326,A -85,B 0,C 180,E1 -1298.481,E2 -1298.481} C_VEL
LIN {X 0,Y 587.308,Z 703.326,A -85,B 0,C 180,E1 -1301.16,E2 -1301.16} C_VEL
LIN {X 0,Y 587.303,Z 703.322,A -85,B 0,C 180,E1 -1304.111,E2 -1304.111} C_VEL
LIN {X 0,Y 587.289,Z 703.334,A -85,B 0,C 180,E1 -1306.991,E2 -1306.991} C_VEL
LIN {X 0,Y 587.292,Z 703.324,A -85,B 0,C 180,E1 -1309.744,E2 -1309.744} C_VEL
LIN {X 0,Y 587.312,Z 703.322,A -85,B 0,C 180,E1 -1312.39,E2 -1312.39} C_VEL
LIN {X 0,Y 587.318,Z 703.322,A -85,B 0,C 180,E1 -1315.657,E2 -1315.657} C_VEL
LIN {X 0,Y 587.318,Z 703.32,A -85,B 0,C 180,E1 -1318.23,E2 -1318.23} C_VEL
LIN {X 0,Y 587.323,Z 703.325,A -85,B 0,C 180,E1 -1320.872,E2 -1320.872} C_VEL
LIN {X 0,Y 587.296,Z 703.325,A -85,B 0,C 180,E1 -1323.833,E2 -1323.833} C_VEL
LIN {X 0,Y 587.299,Z 703.325,A -85,B 0,C 180,E1 -1326.74,E2 -1326.74} C_VEL
LIN {X 0,Y 587.316,Z 703.325,A -85,B 0,C 180,E1 -1329.695,E2 -1329.695} C_VEL
LIN {X 0,Y 587.281,Z 703.328,A -85,B 0,C 180,E1 -1331.872,E2 -1331.872} C_VEL
LIN {X 0,Y 587.296,Z 703.324,A -85,B 0,C 180,E1 -1334.024,E2 -1334.024} C_VEL
LIN {X 0,Y 587.325,Z 703.32,A -85,B 0,C 180,E1 -1336.153,E2 -1336.153} C_VEL
LIN {X 0,Y 587.294,Z 703.325,A -85,B 0,C 180,E1 -1338.962,E2 -1338.962} C_VEL
LIN {X 0,Y 587.32,Z 703.327,A -85,B 0,C 180,E1 -1341.744,E2 -1341.744} C_VEL
LIN {X 0,Y 587.317,Z 703.32,A -85,B 0,C 180,E1 -1344.507,E2 -1344.507} C_VEL
LIN {X 0,Y 587.35,Z 703.32,A -85,B 0,C 180,E1 -1347.257,E2 -1347.257} C_VEL
LIN {X 0,Y 587.382,Z 703.317,A -85,B 0,C 180,E1 -1350,E2 -1350} C_VEL
LIN {X 0,Y 587.34,Z 703.317,A -85,B 0,C 180,E1 -1352.743,E2 -1352.743} C_VEL
LIN {X 0,Y 587.336,Z 703.323,A -85,B 0,C 180,E1 -1355.493,E2 -1355.493} C_VEL
LIN {X 0,Y 587.34,Z 703.321,A -85,B 0,C 180,E1 -1358.256,E2 -1358.256} C_VEL
LIN {X 0,Y 587.335,Z 703.318,A -85,B 0,C 180,E1 -1361.124,E2 -1361.124} C_VEL
LIN {X 0,Y 587.369,Z 703.319,A -85,B 0,C 180,E1 -1364.26,E2 -1364.26} C_VEL
LIN {X 0,Y 587.31,Z 703.323,A -85,B 0,C 180,E1 -1367.407,E2 -1367.407} C_VEL
LIN {X 0,Y 587.31,Z 703.324,A -85,B 0,C 180,E1 -1369.576,E2 -1369.576} C_VEL
LIN {X 0,Y 587.318,Z 703.325,A -85,B 0,C 180,E1 -1371.775,E2 -1371.775} C_VEL
LIN {X 0,Y 587.32,Z 703.321,A -85,B 0,C 180,E1 -1374.76,E2 -1374.76} C_VEL
LIN {X 0,Y 587.305,Z 703.324,A -85,B 0,C 180,E1 -1377.683,E2 -1377.683} C_VEL
LIN {X 0,Y 587.322,Z 703.329,A -85,B 0,C 180,E1 -1380.171,E2 -1380.171} C_VEL
LIN {X 0,Y 587.341,Z 703.322,A -85,B 0,C 180,E1 -1382.579,E2 -1382.579} C_VEL
LIN {X 0,Y 587.328,Z 703.319,A -85,B 0,C 180,E1 -1385.056,E2 -1385.056} C_VEL
LIN {X 0,Y 587.339,Z 703.32,A -85,B 0,C 180,E1 -1387.838,E2 -1387.838} C_VEL
LIN {X 0,Y 587.313,Z 703.329,A -85,B 0,C 180,E1 -1390.255,E2 -1390.255} C_VEL
LIN {X 0,Y 587.321,Z 703.32,A -85,B 0,C 180,E1 -1393.118,E2 -1393.118} C_VEL
LIN {X 0,Y 587.316,Z 703.323,A -85,B 0,C 180,E1 -1396.048,E2 -1396.048} C_VEL
LIN {X 0,Y 587.339,Z 703.323,A -85,B 0,C 180,E1 -1398.925,E2 -1398.925} C_VEL
LIN {X 0,Y 587.363,Z 703.321,A -85,B 0,C 180,E1 -1400.314,E2 -1400.314} C_VEL
LIN {X 0,Y 587.623,Z 706.59,A -85,B 0,C 180,E1 -1400.441,E2 -1400.441} C_VEL
LIN {X 0,Y 587.553,Z 719.231,A -85,B 0,C 180,E1 -1400.964,E2 -1400.964} C_VEL
LIN {X 0,Y 587.458,Z 731.244,A -85,B 0,C 180,E1 -1401.625,E2 -1401.625} C_VEL
LIN {X 0,Y 587.417,Z 740.692,A -85,B 0,C 180,E1 -1402.275,E2 -1402.275} C_VEL
LIN {X 0,Y 587.359,Z 749.869,A -85,B 0,C 180,E1 -1403.039,E2 -1403.039} C_VEL
LIN {X 0,Y 587.3,Z 758.301,A -85,B 0,C 180,E1 -1403.888,E2 -1403.888} C_VEL
LIN {X 0,Y 587.28,Z 765.064,A -85,B 0,C 180,E1 -1404.706,E2 -1404.706} C_VEL
LIN {X 0,Y 587.204,Z 772.332,A -85,B 0,C 180,E1 -1405.769,E2 -1405.769} C_VEL
LIN {X 0,Y 587.168,Z 778.468,A -85,B 0,C 180,E1 -1406.915,E2 -1406.915} C_VEL
LIN {X 0,Y 587.151,Z 783.705,A -85,B 0,C 180,E1 -1408.219,E2 -1408.219} C_VEL
LIN {X 0,Y 587.158,Z 787.277,A -85,B 0,C 180,E1 -1409.521,E2 -1409.521} C_VEL
LIN {X 0,Y 587.167,Z 789.439,A -85,B 0,C 180,E1 -1410.899,E2 -1410.899} C_VEL
LIN {X 0,Y 587.158,Z 789.938,A -85,B 0,C 180,E1 -1412.344,E2 -1412.344} C_VEL
LIN {X 0,Y 587.132,Z 789.64,A -85,B 0,C 180,E1 -1412.944,E2 -1412.944} C_VEL
LIN {X 0,Y 587.12,Z 788.58,A -85,B 0,C 180,E1 -1413.868,E2 -1413.868} C_VEL
LIN {X 0,Y 587.173,Z 785.671,A -85,B 0,C 180,E1 -1415.233,E2 -1415.233} C_VEL
LIN {X 0,Y 587.175,Z 781.956,A -85,B 0,C 180,E1 -1416.361,E2 -1416.361} C_VEL
LIN {X 0,Y 587.182,Z 776.97,A -85,B 0,C 180,E1 -1417.48,E2 -1417.48} C_VEL
LIN {X 0,Y 587.227,Z 770.608,A -85,B 0,C 180,E1 -1418.591,E2 -1418.591} C_VEL
LIN {X 0,Y 587.274,Z 764.096,A -85,B 0,C 180,E1 -1419.51,E2 -1419.51} C_VEL
LIN {X 0,Y 587.314,Z 756.249,A -85,B 0,C 180,E1 -1420.424,E2 -1420.424} C_VEL
LIN {X 0,Y 587.363,Z 746.74,A -85,B 0,C 180,E1 -1421.333,E2 -1421.333} C_VEL
LIN {X 0,Y 587.435,Z 736.113,A -85,B 0,C 180,E1 -1422.147,E2 -1422.147} C_VEL
LIN {X 0,Y 587.492,Z 724.767,A -85,B 0,C 180,E1 -1422.841,E2 -1422.841} C_VEL
LIN {X 0,Y 587.568,Z 712.901,A -85,B 0,C 180,E1 -1423.407,E2 -1423.407} C_VEL
LIN {X 0,Y 587.609,Z 704.488,A -85,B 0,C 180,E1 -1423.721,E2 -1423.721} C_VEL
LIN {X 0,Y 587.352,Z 703.323,A -85,B 0,C 180,E1 -1423.78,E2 -1423.78} C_VEL
LIN {X 0,Y 587.361,Z 703.317,A -85,B 0,C 180,E1 -1426.154,E2 -1426.154} C_VEL
LIN {X 0,Y 587.342,Z 703.319,A -85,B 0,C 180,E1 -1428.962,E2 -1428.962} C_VEL
LIN {X 0,Y 587.366,Z 703.324,A -85,B 0,C 180,E1 -1431.745,E2 -1431.745} C_VEL
LIN {X 0,Y 587.347,Z 703.316,A -85,B 0,C 180,E1 -1434.507,E2 -1434.507} C_VEL
LIN {X 0,Y 587.361,Z 703.317,A -85,B 0,C 180,E1 -1437.257,E2 -1437.257} C_VEL
LIN {X 0,Y 587.39,Z 703.318,A -85,B 0,C 180,E1 -1440,E2 -1440} C_VEL
LIN {X 0,Y 587.376,Z 703.312,A -85,B 0,C 180,E1 -1442.743,E2 -1442.743} C_VEL
LIN {X 0,Y 587.348,Z 703.32,A -85,B 0,C 180,E1 -1445.493,E2 -1445.493} C_VEL
LIN {X 0,Y 587.35,Z 703.32,A -85,B 0,C 180,E1 -1447.563,E2 -1447.563} C_VEL
LIN {X 0,Y 587.345,Z 703.321,A -85,B 0,C 180,E1 -1450.34,E2 -1450.34} C_VEL
LIN {X 0,Y 587.315,Z 703.32,A -85,B 0,C 180,E1 -1453.142,E2 -1453.142} C_VEL
LIN {X 0,Y 587.331,Z 703.318,A -85,B 0,C 180,E1 -1455.263,E2 -1455.263} C_VEL
LIN {X 0,Y 587.351,Z 703.316,A -85,B 0,C 180,E1 -1457.406,E2 -1457.406} C_VEL
LIN {X 0,Y 587.333,Z 703.326,A -85,B 0,C 180,E1 -1460.305,E2 -1460.305} C_VEL
LIN {X 0,Y 587.317,Z 703.32,A -85,B 0,C 180,E1 -1463.259,E2 -1463.259} C_VEL
LIN {X 0,Y 587.332,Z 703.319,A -85,B 0,C 180,E1 -1465.517,E2 -1465.517} C_VEL
LIN {X 0,Y 587.351,Z 703.318,A -85,B 0,C 180,E1 -1467.818,E2 -1467.818} C_VEL
LIN {X 0,Y 587.34,Z 703.326,A -85,B 0,C 180,E1 -1470.51,E2 -1470.51} C_VEL
LIN {X 0,Y 587.338,Z 703.317,A -85,B 0,C 180,E1 -1473.397,E2 -1473.397} C_VEL
LIN {X 0,Y 587.297,Z 703.325,A -85,B 0,C 180,E1 -1475.9,E2 -1475.9} C_VEL
LIN {X 0,Y 587.334,Z 703.328,A -85,B 0,C 180,E1 -1478.479,E2 -1478.479} C_VEL
LIN {X 0,Y 587.34,Z 703.32,A -85,B 0,C 180,E1 -1481.157,E2 -1481.157} C_VEL
LIN {X 0,Y 587.33,Z 703.321,A -85,B 0,C 180,E1 -1484.113,E2 -1484.113} C_VEL
LIN {X 0,Y 587.32,Z 703.326,A -85,B 0,C 180,E1 -1486.994,E2 -1486.994} C_VEL
LIN {X 0,Y 587.319,Z 703.322,A -85,B 0,C 180,E1 -1489.746,E2 -1489.746} C_VEL
LIN {X 0,Y 587.349,Z 703.323,A -85,B 0,C 180,E1 -1492.392,E2 -1492.392} C_VEL
LIN {X 0,Y 587.383,Z 703.511,A -85,B 0,C 180,E1 -1493.575,E2 -1493.575} C_VEL
LIN {X 0,Y 588.002,Z 707.423,A -85,B 0,C 180,E1 -1494.367,E2 -1494.367} C_VEL
LIN {X 0,Y 588.133,Z 721.73,A -85,B 0,C 180,E1 -1497.121,E2 -1497.121} C_VEL
LIN {X 0,Y 587.983,Z 735.147,A -85,B 0,C 180,E1 -1499.866,E2 -1499.866} C_VEL
LIN {X 0,Y 587.81,Z 750.798,A -85,B 0,C 180,E1 -1502.977,E2 -1502.977} C_VEL
LIN {X 0,Y 587.704,Z 764.71,A -85,B 0,C 180,E1 -1505.675,E2 -1505.675} C_VEL
LIN {X 0,Y 587.61,Z 778.188,A -85,B 0,C 180,E1 -1508.237,E2 -1508.237} C_VEL
LIN {X 0,Y 587.492,Z 793.839,A -85,B 0,C 180,E1 -1511.156,E2 -1511.156} C_VEL
LIN {X 0,Y 587.383,Z 809.491,A -85,B 0,C 180,E1 -1514.026,E2 -1514.026} C_VEL
LIN {X 0,Y 587.292,Z 825.142,A -85,B 0,C 180,E1 -1516.858,E2 -1516.858} C_VEL
LIN {X 0,Y 587.314,Z 830.156,A -85,B 0,C 180,E1 -1517.759,E2 -1517.759} C_VEL
LIN {X 0,Y 587.742,Z 835.939,A -85,B 0,C 180,E1 -1517.855,E2 -1517.855} C_VEL
LIN {X 0,Y 587.686,Z 849.213,A -85,B 0,C 180,E1 -1518.161,E2 -1518.161} C_VEL
LIN {X 0,Y 587.623,Z 861.733,A -85,B 0,C 180,E1 -1518.589,E2 -1518.589} C_VEL
LIN {X 0,Y 587.521,Z 873.63,A -85,B 0,C 180,E1 -1519.14,E2 -1519.14} C_VEL
LIN {X 0,Y 587.456,Z 885.198,A -85,B 0,C 180,E1 -1519.836,E2 -1519.836} C_VEL
LIN {X 0,Y 587.367,Z 895.595,A -85,B 0,C 180,E1 -1520.617,E2 -1520.617} C_VEL
LIN {X 0,Y 587.322,Z 904.111,A -85,B 0,C 180,E1 -1521.397,E2 -1521.397} C_VEL
LIN {X 0,Y 587.274,Z 911.959,A -85,B 0,C 180,E1 -1522.263,E2 -1522.263} C_VEL
LIN {X 0,Y 587.23,Z 918.469,A -85,B 0,C 180,E1 -1523.126,E2 -1523.126} C_VEL
LIN {X 0,Y 587.236,Z 924.866,A -85,B 0,C 180,E1 -1524.161,E2 -1524.161} C_VEL
LIN {X 0,Y 587.147,Z 929.95,A -85,B 0,C 180,E1 -1525.194,E2 -1525.194} C_VEL
LIN {X 0,Y 587.212,Z 933.896,A -85,B 0,C 180,E1 -1526.226,E2 -1526.226} C_VEL
LIN {X 0,Y 587.132,Z 936.809,A -85,B 0,C 180,E1 -1527.256,E2 -1527.256} C_VEL
LIN {X 0,Y 587.138,Z 938.201,A -85,B 0,C 180,E1 -1527.942,E2 -1527.942} C_VEL
LIN {X 0,Y 587.14,Z 939.784,A -85,B 0,C 180,E1 -1529.314,E2 -1529.314} C_VEL
LIN {X 0,Y 587.137,Z 940,A -85,B 0,C 180,E1 -1530,E2 -1530} C_VEL
LIN {X 0,Y 587.147,Z 939.185,A -85,B 0,C 180,E1 -1531.372,E2 -1531.372} C_VEL
LIN {X 0,Y 587.138,Z 938.202,A -85,B 0,C 180,E1 -1532.058,E2 -1532.058} C_VEL
LIN {X 0,Y 587.132,Z 936.81,A -85,B 0,C 180,E1 -1532.744,E2 -1532.744} C_VEL
LIN {X 0,Y 587.212,Z 933.896,A -85,B 0,C 180,E1 -1533.774,E2 -1533.774} C_VEL
LIN {X 0,Y 587.147,Z 929.95,A -85,B 0,C 180,E1 -1534.806,E2 -1534.806} C_VEL
LIN {X 0,Y 587.217,Z 923.878,A -85,B 0,C 180,E1 -1536.011,E2 -1536.011} C_VEL
LIN {X 0,Y 587.245,Z 917.236,A -85,B 0,C 180,E1 -1537.046,E2 -1537.046} C_VEL
LIN {X 0,Y 587.299,Z 908.99,A -85,B 0,C 180,E1 -1538.083,E2 -1538.083} C_VEL
LIN {X 0,Y 587.343,Z 900.537,A -85,B 0,C 180,E1 -1538.949,E2 -1538.949} C_VEL
LIN {X 0,Y 587.414,Z 890.094,A -85,B 0,C 180,E1 -1539.816,E2 -1539.816} C_VEL
LIN {X 0,Y 587.504,Z 879.759,A -85,B 0,C 180,E1 -1540.511,E2 -1540.511} C_VEL
LIN {X 0,Y 587.537,Z 868.082,A -85,B 0,C 180,E1 -1541.137,E2 -1541.137} C_VEL
LIN {X 0,Y 587.628,Z 855.651,A -85,B 0,C 180,E1 -1541.637,E2 -1541.637} C_VEL
LIN {X 0,Y 587.71,Z 842.437,A -85,B 0,C 180,E1 -1542.014,E2 -1542.014} C_VEL
LIN {X 0,Y 587.518,Z 831.601,A -85,B 0,C 180,E1 -1542.215,E2 -1542.215} C_VEL
LIN {X 0,Y 587.319,Z 830.034,A -85,B 0,C 180,E1 -1542.263,E2 -1542.263} C_VEL
LIN {X 0,Y 587.38,Z 813.405,A -85,B 0,C 180,E1 -1545.262,E2 -1545.262} C_VEL
LIN {X 0,Y 587.465,Z 797.753,A -85,B 0,C 180,E1 -1548.122,E2 -1548.122} C_VEL
LIN {X 0,Y 587.561,Z 784.058,A -85,B 0,C 180,E1 -1550.662,E2 -1550.662} C_VEL
LIN {X 0,Y 587.645,Z 770.363,A -85,B 0,C 180,E1 -1553.245,E2 -1553.245} C_VEL
LIN {X 0,Y 587.773,Z 756.668,A -85,B 0,C 180,E1 -1555.876,E2 -1555.876} C_VEL
LIN {X 0,Y 587.874,Z 742.973,A -85,B 0,C 180,E1 -1558.568,E2 -1558.568} C_VEL
LIN {X 0,Y 588.017,Z 731.235,A -85,B 0,C 180,E1 -1560.927,E2 -1560.927} C_VEL
LIN {X 0,Y 588.124,Z 718.373,A -85,B 0,C 180,E1 -1563.551,E2 -1563.551} C_VEL
LIN {X 0,Y 588.056,Z 706.875,A -85,B 0,C 180,E1 -1565.846,E2 -1565.846} C_VEL
LIN {X 0,Y 587.368,Z 703.323,A -85,B 0,C 180,E1 -1566.647,E2 -1566.647} C_VEL
LIN {X 0,Y 587.338,Z 703.327,A -85,B 0,C 180,E1 -1569.36,E2 -1569.36} C_VEL
LIN {X 0,Y 587.338,Z 703.318,A -85,B 0,C 180,E1 -1572.108,E2 -1572.108} C_VEL
LIN {X 0,Y 587.32,Z 703.326,A -85,B 0,C 180,E1 -1575.089,E2 -1575.089} C_VEL
LIN {X 0,Y 587.326,Z 703.321,A -85,B 0,C 180,E1 -1577.925,E2 -1577.925} C_VEL
LIN {X 0,Y 587.348,Z 703.316,A -85,B 0,C 180,E1 -1580.641,E2 -1580.641} C_VEL
LIN {X 0,Y 587.35,Z 703.323,A -85,B 0,C 180,E1 -1583.293,E2 -1583.293} C_VEL
LIN {X 0,Y 587.369,Z 703.32,A -85,B 0,C 180,E1 -1585.78,E2 -1585.78} C_VEL
LIN {X 0,Y 587.344,Z 703.318,A -85,B 0,C 180,E1 -1588.231,E2 -1588.231} C_VEL
LIN {X 0,Y 587.353,Z 703.316,A -85,B 0,C 180,E1 -1590.867,E2 -1590.867} C_VEL
LIN {X 0,Y 587.359,Z 703.323,A -85,B 0,C 180,E1 -1593.82,E2 -1593.82} C_VEL
LIN {X 0,Y 587.33,Z 703.324,A -85,B 0,C 180,E1 -1595.993,E2 -1595.993} C_VEL
LIN {X 0,Y 587.322,Z 703.322,A -85,B 0,C 180,E1 -1598.226,E2 -1598.226} C_VEL
LIN {X 0,Y 587.352,Z 703.317,A -85,B 0,C 180,E1 -1601.151,E2 -1601.151} C_VEL
LIN {X 0,Y 587.323,Z 703.327,A -85,B 0,C 180,E1 -1604.025,E2 -1604.025} C_VEL
LIN {X 0,Y 587.356,Z 703.321,A -85,B 0,C 180,E1 -1606.154,E2 -1606.154} C_VEL
LIN {X 0,Y 587.346,Z 703.316,A -85,B 0,C 180,E1 -1608.963,E2 -1608.963} C_VEL
LIN {X 0,Y 587.367,Z 703.32,A -85,B 0,C 180,E1 -1611.745,E2 -1611.745} C_VEL
LIN {X 0,Y 587.344,Z 703.32,A -85,B 0,C 180,E1 -1614.507,E2 -1614.507} C_VEL
LIN {X 0,Y 587.371,Z 703.314,A -85,B 0,C 180,E1 -1617.257,E2 -1617.257} C_VEL
LIN {X 0,Y 587.389,Z 703.32,A -85,B 0,C 180,E1 -1620,E2 -1620} C_VEL
LIN {X 0,Y 587.357,Z 703.317,A -85,B 0,C 180,E1 -1622.743,E2 -1622.743} C_VEL
LIN {X 0,Y 587.345,Z 703.317,A -85,B 0,C 180,E1 -1625.493,E2 -1625.493} C_VEL
LIN {X 0,Y 587.364,Z 703.325,A -85,B 0,C 180,E1 -1628.255,E2 -1628.255} C_VEL
LIN {X 0,Y 587.334,Z 703.318,A -85,B 0,C 180,E1 -1631.124,E2 -1631.124} C_VEL
LIN {X 0,Y 587.353,Z 703.318,A -85,B 0,C 180,E1 -1633.846,E2 -1633.846} C_VEL
LIN {X 0,Y 587.332,Z 703.322,A -85,B 0,C 180,E1 -1636.808,E2 -1636.808} C_VEL
LIN {X 0,Y 587.298,Z 703.327,A -85,B 0,C 180,E1 -1638.291,E2 -1638.291} C_VEL
LIN {X 0,Y 586.657,Z 703.407,A -85,B 0,C 180,E1 -1638.863,E2 -1638.863} C_VEL
LIN {X 0,Y 583.841,Z 703.755,A -85,B 0,C 180,E1 -1639.791,E2 -1639.791} C_VEL
LIN {X 0,Y 581.437,Z 704.063,A -85,B 0,C 180,E1 -1640.539,E2 -1640.539} C_VEL
LIN {X 0,Y 580.383,Z 704.186,A -85,B 0,C 180,E1 -1641.115,E2 -1641.115} C_VEL
LIN {X 0,Y 580.286,Z 704.196,A -85,B 0,C 180,E1 -1641.31,E2 -1641.31} C_VEL
LIN {X 0,Y 580.265,Z 704.199,A -85,B 0,C 180,E1 -1643.559,E2 -1643.559} C_VEL
LIN {X 0,Y 580.259,Z 704.206,A -85,B 0,C 180,E1 -1646.327,E2 -1646.327} C_VEL
LIN {X 0,Y 580.276,Z 704.199,A -85,B 0,C 180,E1 -1649.305,E2 -1649.305} C_VEL
LIN {X 0,Y 580.299,Z 704.198,A -85,B 0,C 180,E1 -1652.201,E2 -1652.201} C_VEL
LIN {X 0,Y 580.282,Z 704.206,A -85,B 0,C 180,E1 -1654.697,E2 -1654.697} C_VEL
LIN {X 0,Y 580.269,Z 704.201,A -85,B 0,C 180,E1 -1657.271,E2 -1657.271} C_VEL
LIN {X 0,Y 580.28,Z 704.199,A -85,B 0,C 180,E1 -1660.269,E2 -1660.269} C_VEL
LIN {X 0,Y 580.236,Z 704.205,A -85,B 0,C 180,E1 -1663.386,E2 -1663.386} C_VEL
LIN {X 0,Y 580.238,Z 704.204,A -85,B 0,C 180,E1 -1666.338,E2 -1666.338} C_VEL
LIN {X 0,Y 580.256,Z 704.208,A -85,B 0,C 180,E1 -1669.153,E2 -1669.153} C_VEL
LIN {X 0,Y 580.276,Z 704.198,A -85,B 0,C 180,E1 -1671.929,E2 -1671.929} C_VEL
LIN {X 0,Y 580.224,Z 704.206,A -85,B 0,C 180,E1 -1674.451,E2 -1674.451} C_VEL
LIN {X 0,Y 580.239,Z 704.21,A -85,B 0,C 180,E1 -1676.972,E2 -1676.972} C_VEL
LIN {X 0,Y 580.268,Z 704.205,A -85,B 0,C 180,E1 -1679.423,E2 -1679.423} C_VEL
LIN {X 0,Y 580.24,Z 704.202,A -85,B 0,C 180,E1 -1682.153,E2 -1682.153} C_VEL
LIN {X 0,Y 580.231,Z 704.208,A -85,B 0,C 180,E1 -1684.917,E2 -1684.917} C_VEL
LIN {X 0,Y 580.284,Z 704.206,A -85,B 0,C 180,E1 -1687.197,E2 -1687.197} C_VEL
LIN {X 0,Y 580.268,Z 704.208,A -85,B 0,C 180,E1 -1689.437,E2 -1689.437} C_VEL
LIN {X 0,Y 580.242,Z 704.208,A -85,B 0,C 180,E1 -1691.644,E2 -1691.644} C_VEL
LIN {X 0,Y 580.254,Z 704.204,A -85,B 0,C 180,E1 -1693.825,E2 -1693.825} C_VEL
LIN {X 0,Y 580.291,Z 704.198,A -85,B 0,C 180,E1 -1695.982,E2 -1695.982} C_VEL
LIN {X 0,Y 580.271,Z 704.199,A -85,B 0,C 180,E1 -1698.826,E2 -1698.826} C_VEL
LIN {X 0,Y 580.292,Z 704.205,A -85,B 0,C 180,E1 -1701.643,E2 -1701.643} C_VEL
LIN {X 0,Y 580.287,Z 704.196,A -85,B 0,C 180,E1 -1704.44,E2 -1704.44} C_VEL
LIN {X 0,Y 580.316,Z 704.196,A -85,B 0,C 180,E1 -1707.223,E2 -1707.223} C_VEL
LIN {X 0,Y 580.351,Z 704.193,A -85,B 0,C 180,E1 -1710,E2 -1710} C_VEL
LIN {X 0,Y 580.308,Z 704.193,A -85,B 0,C 180,E1 -1712.777,E2 -1712.777} C_VEL
LIN {X 0,Y 580.305,Z 704.2,A -85,B 0,C 180,E1 -1715.56,E2 -1715.56} C_VEL
LIN {X 0,Y 580.308,Z 704.196,A -85,B 0,C 180,E1 -1718.356,E2 -1718.356} C_VEL
LIN {X 0,Y 580.306,Z 704.194,A -85,B 0,C 180,E1 -1721.191,E2 -1721.191} C_VEL
LIN {X 0,Y 580.325,Z 704.2,A -85,B 0,C 180,E1 -1724.017,E2 -1724.017} C_VEL
LIN {X 0,Y 580.295,Z 704.195,A -85,B 0,C 180,E1 -1726.906,E2 -1726.906} C_VEL
LIN {X 0,Y 580.286,Z 704.203,A -85,B 0,C 180,E1 -1729.823,E2 -1729.823} C_VEL
LIN {X 0,Y 580.271,Z 704.208,A -85,B 0,C 180,E1 -1732.053,E2 -1732.053} C_VEL
LIN {X 0,Y 580.288,Z 704.195,A -85,B 0,C 180,E1 -1735.081,E2 -1735.081} C_VEL
LIN {X 0,Y 580.285,Z 704.207,A -85,B 0,C 180,E1 -1738.187,E2 -1738.187} C_VEL
LIN {X 0,Y 580.28,Z 704.2,A -85,B 0,C 180,E1 -1740.693,E2 -1740.693} C_VEL
LIN {X 0,Y 580.284,Z 704.196,A -85,B 0,C 180,E1 -1743.313,E2 -1743.313} C_VEL
LIN {X 0,Y 580.248,Z 704.203,A -85,B 0,C 180,E1 -1745.756,E2 -1745.756} C_VEL
LIN {X 0,Y 580.29,Z 704.202,A -85,B 0,C 180,E1 -1748.147,E2 -1748.147} C_VEL
LIN {X 0,Y 580.3,Z 704.198,A -85,B 0,C 180,E1 -1750.844,E2 -1750.844} C_VEL
LIN {X 0,Y 580.277,Z 704.197,A -85,B 0,C 180,E1 -1753.658,E2 -1753.658} C_VEL
LIN {X 0,Y 580.278,Z 704.207,A -85,B 0,C 180,E1 -1756.61,E2 -1756.61} C_VEL
LIN {X 0,Y 580.302,Z 704.197,A -85,B 0,C 180,E1 -1759.157,E2 -1759.157} C_VEL
LIN {X 0,Y 580.329,Z 704.331,A -85,B 0,C 180,E1 -1760.217,E2 -1760.217} C_VEL
LIN {X 0,Y 580.651,Z 709.59,A -85,B 0,C 180,E1 -1760.41,E2 -1760.41} C_VEL
LIN {X 0,Y 580.593,Z 721.023,A -85,B 0,C 180,E1 -1760.92,E2 -1760.92} C_VEL
LIN {X 0,Y 580.456,Z 731.802,A -85,B 0,C 180,E1 -1761.535,E2 -1761.535} C_VEL
LIN {X 0,Y 580.399,Z 741.304,A -85,B 0,C 180,E1 -1762.204,E2 -1762.204} C_VEL
LIN {X 0,Y 580.328,Z 749.855,A -85,B 0,C 180,E1 -1762.929,E2 -1762.929} C_VEL
LIN {X 0,Y 580.264,Z 758.164,A -85,B 0,C 180,E1 -1763.775,E2 -1763.775} C_VEL
LIN {X 0,Y 580.223,Z 765.414,A -85,B 0,C 180,E1 -1764.663,E2 -1764.663} C_VEL
LIN {X 0,Y 580.146,Z 771.916,A -85,B 0,C 180,E1 -1765.627,E2 -1765.627} C_VEL
LIN {X 0,Y 580.095,Z 777.838,A -85,B 0,C 180,E1 -1766.716,E2 -1766.716} C_VEL
LIN {X 0,Y 580.069,Z 783.15,A -85,B 0,C 180,E1 -1768.007,E2 -1768.007} C_VEL
LIN {X 0,Y 580.069,Z 786.941,A -85,B 0,C 180,E1 -1769.342,E2 -1769.342} C_VEL
LIN {X 0,Y 580.052,Z 788.602,A -85,B 0,C 180,E1 -1770.214,E2 -1770.214} C_VEL
LIN {X 0,Y 580.058,Z 789.557,A -85,B 0,C 180,E1 -1771.011,E2 -1771.011} C_VEL
LIN {X 0,Y 580.048,Z 789.974,A -85,B 0,C 180,E1 -1772.189,E2 -1772.189} C_VEL
LIN {X 0,Y 580.047,Z 788.816,A -85,B 0,C 180,E1 -1773.716,E2 -1773.716} C_VEL
LIN {X 0,Y 580.045,Z 786.585,A -85,B 0,C 180,E1 -1774.908,E2 -1774.908} C_VEL
LIN {X 0,Y 580.092,Z 783.251,A -85,B 0,C 180,E1 -1776.055,E2 -1776.055} C_VEL
LIN {X 0,Y 580.1,Z 778.697,A -85,B 0,C 180,E1 -1777.189,E2 -1777.189} C_VEL
LIN {X 0,Y 580.134,Z 772.814,A -85,B 0,C 180,E1 -1778.316,E2 -1778.316} C_VEL
LIN {X 0,Y 580.223,Z 765.349,A -85,B 0,C 180,E1 -1779.435,E2 -1779.435} C_VEL
LIN {X 0,Y 580.273,Z 757.748,A -85,B 0,C 180,E1 -1780.361,E2 -1780.361} C_VEL
LIN {X 0,Y 580.298,Z 750.548,A -85,B 0,C 180,E1 -1781.097,E2 -1781.097} C_VEL
LIN {X 0,Y 580.39,Z 741.998,A -85,B 0,C 180,E1 -1781.832,E2 -1781.832} C_VEL
LIN {X 0,Y 580.468,Z 731.68,A -85,B 0,C 180,E1 -1782.563,E2 -1782.563} C_VEL
LIN {X 0,Y 580.532,Z 720.46,A -85,B 0,C 180,E1 -1783.2,E2 -1783.2} C_VEL
LIN {X 0,Y 580.625,Z 707.925,A -85,B 0,C 180,E1 -1783.745,E2 -1783.745} C_VEL
LIN {X 0,Y 580.311,Z 704.198,A -85,B 0,C 180,E1 -1783.894,E2 -1783.894} C_VEL
LIN {X 0,Y 580.332,Z 704.195,A -85,B 0,C 180,E1 -1785.983,E2 -1785.983} C_VEL
LIN {X 0,Y 580.311,Z 704.194,A -85,B 0,C 180,E1 -1788.827,E2 -1788.827} C_VEL
LIN {X 0,Y 580.328,Z 704.202,A -85,B 0,C 180,E1 -1791.644,E2 -1791.644} C_VEL
LIN {X 0,Y 580.314,Z 704.193,A -85,B 0,C 180,E1 -1794.44,E2 -1794.44} C_VEL
LIN {X 0,Y 580.329,Z 704.193,A -85,B 0,C 180,E1 -1797.223,E2 -1797.223} C_VEL
LIN {X 0,Y 580.359,Z 704.194,A -85,B 0,C 180,E1 -1800,E2 -1800} C_VEL
LIN {X 0,Y 580.342,Z 704.188,A -85,B 0,C 180,E1 -1802.776,E2 -1802.776} C_VEL
LIN {X 0,Y 580.316,Z 704.197,A -85,B 0,C 180,E1 -1805.56,E2 -1805.56} C_VEL
LIN {X 0,Y 580.316,Z 704.197,A -85,B 0,C 180,E1 -1807.655,E2 -1807.655} C_VEL
LIN {X 0,Y 580.305,Z 704.197,A -85,B 0,C 180,E1 -1810.467,E2 -1810.467} C_VEL
LIN {X 0,Y 580.272,Z 704.198,A -85,B 0,C 180,E1 -1813.304,E2 -1813.304} C_VEL
LIN {X 0,Y 580.296,Z 704.195,A -85,B 0,C 180,E1 -1815.453,E2 -1815.453} C_VEL
LIN {X 0,Y 580.295,Z 704.197,A -85,B 0,C 180,E1 -1817.624,E2 -1817.624} C_VEL
LIN {X 0,Y 580.292,Z 704.2,A -85,B 0,C 180,E1 -1819.823,E2 -1819.823} C_VEL
LIN {X 0,Y 580.275,Z 704.204,A -85,B 0,C 180,E1 -1822.053,E2 -1822.053} C_VEL
LIN {X 0,Y 580.308,Z 704.194,A -85,B 0,C 180,E1 -1825.08,E2 -1825.08} C_VEL
LIN {X 0,Y 580.304,Z 704.202,A -85,B 0,C 180,E1 -1828.185,E2 -1828.185} C_VEL
LIN {X 0,Y 580.288,Z 704.201,A -85,B 0,C 180,E1 -1830.694,E2 -1830.694} C_VEL
LIN {X 0,Y 580.308,Z 704.193,A -85,B 0,C 180,E1 -1833.316,E2 -1833.316} C_VEL
LIN {X 0,Y 580.253,Z 704.201,A -85,B 0,C 180,E1 -1835.757,E2 -1835.757} C_VEL
LIN {X 0,Y 580.291,Z 704.2,A -85,B 0,C 180,E1 -1838.146,E2 -1838.146} C_VEL
LIN {X 0,Y 580.303,Z 704.201,A -85,B 0,C 180,E1 -1840.843,E2 -1840.843} C_VEL
LIN {X 0,Y 580.283,Z 704.197,A -85,B 0,C 180,E1 -1843.658,E2 -1843.658} C_VEL
LIN {X 0,Y 580.282,Z 704.207,A -85,B 0,C 180,E1 -1846.609,E2 -1846.609} C_VEL
LIN {X 0,Y 580.304,Z 704.2,A -85,B 0,C 180,E1 -1849.157,E2 -1849.157} C_VEL
LIN {X 0,Y 580.294,Z 704.199,A -85,B 0,C 180,E1 -1851.927,E2 -1851.927} C_VEL
LIN {X 0,Y 580.337,Z 704.26,A -85,B 0,C 180,E1 -1853.362,E2 -1853.362} C_VEL
LIN {X 0,Y 581.032,Z 707.941,A -85,B 0,C 180,E1 -1854.137,E2 -1854.137} C_VEL
LIN {X 0,Y 581.198,Z 721.722,A -85,B 0,C 180,E1 -1856.792,E2 -1856.792} C_VEL
LIN {X 0,Y 581.182,Z 729.277,A -85,B 0,C 180,E1 -1858.262,E2 -1858.262} C_VEL
LIN {X 0,Y 581.02,Z 741.723,A -85,B 0,C 180,E1 -1860.81,E2 -1860.81} C_VEL
LIN {X 0,Y 580.877,Z 755.439,A -85,B 0,C 180,E1 -1863.55,E2 -1863.55} C_VEL
LIN {X 0,Y 580.68,Z 770.362,A -85,B 0,C 180,E1 -1866.459,E2 -1866.459} C_VEL
LIN {X 0,Y 580.575,Z 786.014,A -85,B 0,C 180,E1 -1869.448,E2 -1869.448} C_VEL
LIN {X 0,Y 580.42,Z 801.665,A -85,B 0,C 180,E1 -1872.379,E2 -1872.379} C_VEL
LIN {X 0,Y 580.306,Z 817.317,A -85,B 0,C 180,E1 -1875.266,E2 -1875.266} C_VEL
LIN {X 0,Y 580.27,Z 830.156,A -85,B 0,C 180,E1 -1877.608,E2 -1877.608} C_VEL
LIN {X 0,Y 580.824,Z 835.939,A -85,B 0,C 180,E1 -1877.708,E2 -1877.708} C_VEL
LIN {X 0,Y 580.743,Z 849.213,A -85,B 0,C 180,E1 -1878.017,E2 -1878.017} C_VEL
LIN {X 0,Y 580.669,Z 861.367,A -85,B 0,C 180,E1 -1878.436,E2 -1878.436} C_VEL
LIN {X 0,Y 580.544,Z 873.629,A -85,B 0,C 180,E1 -1879.008,E2 -1879.008} C_VEL
LIN {X 0,Y 580.424,Z 885.199,A -85,B 0,C 180,E1 -1879.712,E2 -1879.712} C_VEL
LIN {X 0,Y 580.346,Z 895.595,A -85,B 0,C 180,E1 -1880.503,E2 -1880.503} C_VEL
LIN {X 0,Y 580.271,Z 904.111,A -85,B 0,C 180,E1 -1881.292,E2 -1881.292} C_VEL
LIN {X 0,Y 580.222,Z 911.959,A -85,B 0,C 180,E1 -1882.168,E2 -1882.168} C_VEL
LIN {X 0,Y 580.154,Z 919.649,A -85,B 0,C 180,E1 -1883.222,E2 -1883.222} C_VEL
LIN {X 0,Y 580.139,Z 926.68,A -85,B 0,C 180,E1 -1884.438,E2 -1884.438} C_VEL
LIN {X 0,Y 580.108,Z 931.371,A -85,B 0,C 180,E1 -1885.483,E2 -1885.483} C_VEL
LIN {X 0,Y 580.123,Z 934.956,A -85,B 0,C 180,E1 -1886.527,E2 -1886.527} C_VEL
LIN {X 0,Y 580.043,Z 936.808,A -85,B 0,C 180,E1 -1887.222,E2 -1887.222} C_VEL
LIN {X 0,Y 580.038,Z 938.2,A -85,B 0,C 180,E1 -1887.917,E2 -1887.917} C_VEL
LIN {X 0,Y 580.04,Z 939.784,A -85,B 0,C 180,E1 -1889.306,E2 -1889.306} C_VEL
LIN {X 0,Y 580.037,Z 940,A -85,B 0,C 180,E1 -1890,E2 -1890} C_VEL
LIN {X 0,Y 580.047,Z 939.185,A -85,B 0,C 180,E1 -1891.388,E2 -1891.388} C_VEL
LIN {X 0,Y 580.038,Z 938.201,A -85,B 0,C 180,E1 -1892.083,E2 -1892.083} C_VEL
LIN {X 0,Y 580.043,Z 936.81,A -85,B 0,C 180,E1 -1892.778,E2 -1892.778} C_VEL
LIN {X 0,Y 580.109,Z 933.896,A -85,B 0,C 180,E1 -1893.821,E2 -1893.821} C_VEL
LIN {X 0,Y 580.054,Z 929.95,A -85,B 0,C 180,E1 -1894.865,E2 -1894.865} C_VEL
LIN {X 0,Y 580.139,Z 923.878,A -85,B 0,C 180,E1 -1896.085,E2 -1896.085} C_VEL
LIN {X 0,Y 580.184,Z 917.237,A -85,B 0,C 180,E1 -1897.132,E2 -1897.132} C_VEL
LIN {X 0,Y 580.25,Z 908.99,A -85,B 0,C 180,E1 -1898.182,E2 -1898.182} C_VEL
LIN {X 0,Y 580.308,Z 900.538,A -85,B 0,C 180,E1 -1899.058,E2 -1899.058} C_VEL
LIN {X 0,Y 580.414,Z 890.095,A -85,B 0,C 180,E1 -1899.936,E2 -1899.936} C_VEL
LIN {X 0,Y 580.519,Z 879.759,A -85,B 0,C 180,E1 -1900.639,E2 -1900.639} C_VEL
LIN {X 0,Y 580.573,Z 868.495,A -85,B 0,C 180,E1 -1901.252,E2 -1901.252} C_VEL
LIN {X 0,Y 580.666,Z 856.767,A -85,B 0,C 180,E1 -1901.741,E2 -1901.741} C_VEL
LIN {X 0,Y 580.785,Z 843.351,A -85,B 0,C 180,E1 -1902.137,E2 -1902.137} C_VEL
LIN {X 0,Y 580.632,Z 832.544,A -85,B 0,C 180,E1 -1902.348,E2 -1902.348} C_VEL
LIN {X 0,Y 580.253,Z 830.034,A -85,B 0,C 180,E1 -1902.415,E2 -1902.415} C_VEL
LIN {X 0,Y 580.339,Z 815.361,A -85,B 0,C 180,E1 -1905.092,E2 -1905.092} C_VEL
LIN {X 0,Y 580.44,Z 799.71,A -85,B 0,C 180,E1 -1907.984,E2 -1907.984} C_VEL
LIN {X 0,Y 580.588,Z 784.2,A -85,B 0,C 180,E1 -1910.895,E2 -1910.895} C_VEL
LIN {X 0,Y 580.735,Z 768.407,A -85,B 0,C 180,E1 -1913.917,E2 -1913.917} C_VEL
LIN {X 0,Y 580.886,Z 754.712,A -85,B 0,C 180,E1 -1916.593,E2 -1916.593} C_VEL
LIN {X 0,Y 581.086,Z 739.06,A -85,B 0,C 180,E1 -1919.728,E2 -1919.728} C_VEL
LIN {X 0,Y 581.224,Z 725.209,A -85,B 0,C 180,E1 -1922.553,E2 -1922.553} C_VEL
LIN {X 0,Y 581.219,Z 711.591,A -85,B 0,C 180,E1 -1925.267,E2 -1925.267} C_VEL
LIN {X 0,Y 581.042,Z 707.79,A -85,B 0,C 180,E1 -1926.073,E2 -1926.073} C_VEL
LIN {X 0,Y 580.327,Z 704.201,A -85,B 0,C 180,E1 -1926.875,E2 -1926.875} C_VEL
LIN {X 0,Y 580.289,Z 704.198,A -85,B 0,C 180,E1 -1929.933,E2 -1929.933} C_VEL
LIN {X 0,Y 580.282,Z 704.199,A -85,B 0,C 180,E1 -1932.706,E2 -1932.706} C_VEL
LIN {X 0,Y 580.273,Z 704.204,A -85,B 0,C 180,E1 -1935.609,E2 -1935.609} C_VEL
LIN {X 0,Y 580.283,Z 704.197,A -85,B 0,C 180,E1 -1938.231,E2 -1938.231} C_VEL
LIN {X 0,Y 580.291,Z 704.198,A -85,B 0,C 180,E1 -1940.966,E2 -1940.966} C_VEL
LIN {X 0,Y 580.272,Z 704.206,A -85,B 0,C 180,E1 -1943.597,E2 -1943.597} C_VEL
LIN {X 0,Y 580.322,Z 704.193,A -85,B 0,C 180,E1 -1946.146,E2 -1946.146} C_VEL
LIN {X 0,Y 580.279,Z 704.197,A -85,B 0,C 180,E1 -1948.615,E2 -1948.615} C_VEL
LIN {X 0,Y 580.296,Z 704.196,A -85,B 0,C 180,E1 -1951.024,E2 -1951.024} C_VEL
LIN {X 0,Y 580.293,Z 704.206,A -85,B 0,C 180,E1 -1953.666,E2 -1953.666} C_VEL
LIN {X 0,Y 580.3,Z 704.205,A -85,B 0,C 180,E1 -1955.684,E2 -1955.684} C_VEL
LIN {X 0,Y 580.288,Z 704.196,A -85,B 0,C 180,E1 -1958.695,E2 -1958.695} C_VEL
LIN {X 0,Y 580.302,Z 704.194,A -85,B 0,C 180,E1 -1960.913,E2 -1960.913} C_VEL
LIN {X 0,Y 580.28,Z 704.207,A -85,B 0,C 180,E1 -1963.826,E2 -1963.826} C_VEL
LIN {X 0,Y 580.325,Z 704.2,A -85,B 0,C 180,E1 -1965.983,E2 -1965.983} C_VEL
LIN {X 0,Y 580.309,Z 704.193,A -85,B 0,C 180,E1 -1968.827,E2 -1968.827} C_VEL
LIN {X 0,Y 580.33,Z 704.196,A -85,B 0,C 180,E1 -1971.644,E2 -1971.644} C_VEL
LIN {X 0,Y 580.286,Z 704.202,A -85,B 0,C 180,E1 -1973.742,E2 -1973.742} C_VEL
LIN {X 0,Y 580.274,Z 704.205,A -85,B 0,C 180,E1 -1975.833,E2 -1975.833} C_VEL
LIN {X 0,Y 580.345,Z 704.197,A -85,B 0,C 180,E1 -1977.918,E2 -1977.918} C_VEL
LIN {X 0,Y 580.348,Z 704.19,A -85,B 0,C 180,E1 -1980.694,E2 -1980.694} C_VEL
LIN {X 0,Y 580.325,Z 704.193,A -85,B 0,C 180,E1 -1982.777,E2 -1982.777} C_VEL
LIN {X 0,Y 580.312,Z 704.194,A -85,B 0,C 180,E1 -1985.56,E2 -1985.56} C_VEL
LIN {X 0,Y 580.326,Z 704.2,A -85,B 0,C 180,E1 -1988.356,E2 -1988.356} C_VEL
LIN {X 0,Y 580.304,Z 704.194,A -85,B 0,C 180,E1 -1991.191,E2 -1991.191} C_VEL
LIN {X 0,Y 580.314,Z 704.197,A -85,B 0,C 180,E1 -1994.017,E2 -1994.017} C_VEL
LIN {X 0,Y 580.293,Z 704.198,A -85,B 0,C 180,E1 -1996.906,E2 -1996.906} C_VEL
LIN {X 0,Y 580.284,Z 704.198,A -85,B 0,C 180,E1 -1999.823,E2 -1999.823} C_VEL
LIN {X 0,Y 580.286,Z 704.196,A -85,B 0,C 180,E1 -2001.31,E2 -2001.31} C_VEL
LIN {X 0,Y 579.584,Z 704.286,A -85,B 0,C 180,E1 -2001.889,E2 -2001.889} C_VEL
LIN {X 0,Y 576.704,Z 704.648,A -85,B 0,C 180,E1 -2002.829,E2 -2002.829} C_VEL
LIN {X 0,Y 574.302,Z 704.944,A -85,B 0,C 180,E1 -2003.585,E2 -2003.585} C_VEL
LIN {X 0,Y 573.288,Z 705.072,A -85,B 0,C 180,E1 -2004.169,E2 -2004.169} C_VEL
LIN {X 0,Y 573.214,Z 705.082,A -85,B 0,C 180,E1 -2004.367,E2 -2004.367} C_VEL
LIN {X 0,Y 573.188,Z 705.085,A -85,B 0,C 180,E1 -2006.979,E2 -2006.979} C_VEL
LIN {X 0,Y 573.222,Z 705.077,A -85,B 0,C 180,E1 -2009.483,E2 -2009.483} C_VEL
LIN {X 0,Y 573.252,Z 705.076,A -85,B 0,C 180,E1 -2012.228,E2 -2012.228} C_VEL
LIN {X 0,Y 573.227,Z 705.085,A -85,B 0,C 180,E1 -2014.77,E2 -2014.77} C_VEL
LIN {X 0,Y 573.217,Z 705.077,A -85,B 0,C 180,E1 -2017.809,E2 -2017.809} C_VEL
LIN {X 0,Y 573.248,Z 705.078,A -85,B 0,C 180,E1 -2020.525,E2 -2020.525} C_VEL
LIN {X 0,Y 573.206,Z 705.079,A -85,B 0,C 180,E1 -2023.665,E2 -2023.665} C_VEL
LIN {X 0,Y 573.202,Z 705.084,A -85,B 0,C 180,E1 -2026.637,E2 -2026.637} C_VEL
LIN {X 0,Y 573.231,Z 705.078,A -85,B 0,C 180,E1 -2029.477,E2 -2029.477} C_VEL
LIN {X 0,Y 573.217,Z 705.077,A -85,B 0,C 180,E1 -2032.191,E2 -2032.191} C_VEL
LIN {X 0,Y 573.22,Z 705.085,A -85,B 0,C 180,E1 -2035.232,E2 -2035.232} C_VEL
LIN {X 0,Y 573.221,Z 705.076,A -85,B 0,C 180,E1 -2038.183,E2 -2038.183} C_VEL
LIN {X 0,Y 573.228,Z 705.078,A -85,B 0,C 180,E1 -2040.632,E2 -2040.632} C_VEL
LIN {X 0,Y 573.193,Z 705.086,A -85,B 0,C 180,E1 -2043.517,E2 -2043.517} C_VEL
LIN {X 0,Y 573.198,Z 705.08,A -85,B 0,C 180,E1 -2046.133,E2 -2046.133} C_VEL
LIN {X 0,Y 573.249,Z 705.081,A -85,B 0,C 180,E1 -2049.174,E2 -2049.174} C_VEL
LIN {X 0,Y 573.2,Z 705.088,A -85,B 0,C 180,E1 -2051.41,E2 -2051.41} C_VEL
LIN {X 0,Y 573.224,Z 705.083,A -85,B 0,C 180,E1 -2053.621,E2 -2053.621} C_VEL
LIN {X 0,Y 573.24,Z 705.078,A -85,B 0,C 180,E1 -2055.806,E2 -2055.806} C_VEL
LIN {X 0,Y 573.229,Z 705.076,A -85,B 0,C 180,E1 -2058.765,E2 -2058.765} C_VEL
LIN {X 0,Y 573.237,Z 705.084,A -85,B 0,C 180,E1 -2061.54,E2 -2061.54} C_VEL
LIN {X 0,Y 573.257,Z 705.072,A -85,B 0,C 180,E1 -2064.372,E2 -2064.372} C_VEL
LIN {X 0,Y 573.306,Z 705.072,A -85,B 0,C 180,E1 -2067.892,E2 -2067.892} C_VEL
LIN {X 0,Y 573.32,Z 705.069,A -85,B 0,C 180,E1 -2070,E2 -2070} C_VEL
LIN {X 0,Y 573.276,Z 705.069,A -85,B 0,C 180,E1 -2072.811,E2 -2072.811} C_VEL
LIN {X 0,Y 573.274,Z 705.077,A -85,B 0,C 180,E1 -2075.628,E2 -2075.628} C_VEL
LIN {X 0,Y 573.25,Z 705.074,A -85,B 0,C 180,E1 -2078.46,E2 -2078.46} C_VEL
LIN {X 0,Y 573.277,Z 705.071,A -85,B 0,C 180,E1 -2081.312,E2 -2081.312} C_VEL
LIN {X 0,Y 573.285,Z 705.071,A -85,B 0,C 180,E1 -2084.424,E2 -2084.424} C_VEL
LIN {X 0,Y 573.251,Z 705.072,A -85,B 0,C 180,E1 -2087.112,E2 -2087.112} C_VEL
LIN {X 0,Y 573.242,Z 705.083,A -85,B 0,C 180,E1 -2090.077,E2 -2090.077} C_VEL
LIN {X 0,Y 573.235,Z 705.081,A -85,B 0,C 180,E1 -2092.338,E2 -2092.338} C_VEL
LIN {X 0,Y 573.237,Z 705.075,A -85,B 0,C 180,E1 -2094.871,E2 -2094.871} C_VEL
LIN {X 0,Y 573.239,Z 705.078,A -85,B 0,C 180,E1 -2097.768,E2 -2097.768} C_VEL
LIN {X 0,Y 573.242,Z 705.084,A -85,B 0,C 180,E1 -2100.177,E2 -2100.177} C_VEL
LIN {X 0,Y 573.256,Z 705.076,A -85,B 0,C 180,E1 -2102.645,E2 -2102.645} C_VEL
LIN {X 0,Y 573.209,Z 705.077,A -85,B 0,C 180,E1 -2105.188,E2 -2105.188} C_VEL
LIN {X 0,Y 573.238,Z 705.076,A -85,B 0,C 180,E1 -2107.808,E2 -2107.808} C_VEL
LIN {X 0,Y 573.249,Z 705.081,A -85,B 0,C 180,E1 -2110.525,E2 -2110.525} C_VEL
LIN {X 0,Y 573.242,Z 705.073,A -85,B 0,C 180,E1 -2113.359,E2 -2113.359} C_VEL
LIN {X 0,Y 573.241,Z 705.083,A -85,B 0,C 180,E1 -2116.641,E2 -2116.641} C_VEL
LIN {X 0,Y 573.249,Z 705.074,A -85,B 0,C 180,E1 -2119.475,E2 -2119.475} C_VEL
LIN {X 0,Y 573.26,Z 705.076,A -85,B 0,C 180,E1 -2120.08,E2 -2120.08} C_VEL
LIN {X 0,Y 573.709,Z 709.406,A -85,B 0,C 180,E1 -2120.26,E2 -2120.26} C_VEL
LIN {X 0,Y 573.615,Z 721.708,A -85,B 0,C 180,E1 -2120.82,E2 -2120.82} C_VEL
LIN {X 0,Y 573.46,Z 732.019,A -85,B 0,C 180,E1 -2121.421,E2 -2121.421} C_VEL
LIN {X 0,Y 573.385,Z 741.589,A -85,B 0,C 180,E1 -2122.107,E2 -2122.107} C_VEL
LIN {X 0,Y 573.283,Z 749.995,A -85,B 0,C 180,E1 -2122.831,E2 -2122.831} C_VEL
LIN {X 0,Y 573.196,Z 758.662,A -85,B 0,C 180,E1 -2123.729,E2 -2123.729} C_VEL
LIN {X 0,Y 573.122,Z 767.121,A -85,B 0,C 180,E1 -2124.806,E2 -2124.806} C_VEL
LIN {X 0,Y 573.044,Z 773.799,A -85,B 0,C 180,E1 -2125.868,E2 -2125.868} C_VEL
LIN {X 0,Y 572.998,Z 779.097,A -85,B 0,C 180,E1 -2126.924,E2 -2126.924} C_VEL
LIN {X 0,Y 572.966,Z 783.821,A -85,B 0,C 180,E1 -2128.167,E2 -2128.167} C_VEL
LIN {X 0,Y 572.981,Z 786.607,A -85,B 0,C 180,E1 -2129.16,E2 -2129.16} C_VEL
LIN {X 0,Y 572.95,Z 787.983,A -85,B 0,C 180,E1 -2129.806,E2 -2129.806} C_VEL
LIN {X 0,Y 572.987,Z 789.153,A -85,B 0,C 180,E1 -2130.618,E2 -2130.618} C_VEL
LIN {X 0,Y 572.942,Z 790,A -85,B 0,C 180,E1 -2132.03,E2 -2132.03} C_VEL
LIN {X 0,Y 572.939,Z 789.613,A -85,B 0,C 180,E1 -2133.008,E2 -2133.008} C_VEL
LIN {X 0,Y 572.946,Z 788.731,A -85,B 0,C 180,E1 -2133.794,E2 -2133.794} C_VEL
LIN {X 0,Y 572.961,Z 785.985,A -85,B 0,C 180,E1 -2135.189,E2 -2135.189} C_VEL
LIN {X 0,Y 573.002,Z 781.786,A -85,B 0,C 180,E1 -2136.508,E2 -2136.508} C_VEL
LIN {X 0,Y 572.998,Z 776.761,A -85,B 0,C 180,E1 -2137.652,E2 -2137.652} C_VEL
LIN {X 0,Y 573.084,Z 771.405,A -85,B 0,C 180,E1 -2138.622,E2 -2138.622} C_VEL
LIN {X 0,Y 573.144,Z 765.204,A -85,B 0,C 180,E1 -2139.545,E2 -2139.545} C_VEL
LIN {X 0,Y 573.222,Z 757.573,A -85,B 0,C 180,E1 -2140.482,E2 -2140.482} C_VEL
LIN {X 0,Y 573.275,Z 750.262,A -85,B 0,C 180,E1 -2141.234,E2 -2141.234} C_VEL
LIN {X 0,Y 573.362,Z 741.756,A -85,B 0,C 180,E1 -2141.971,E2 -2141.971} C_VEL
LIN {X 0,Y 573.464,Z 731.39,A -85,B 0,C 180,E1 -2142.711,E2 -2142.711} C_VEL
LIN {X 0,Y 573.597,Z 719.863,A -85,B 0,C 180,E1 -2143.367,E2 -2143.367} C_VEL
LIN {X 0,Y 573.711,Z 707.314,A -85,B 0,C 180,E1 -2143.909,E2 -2143.909} C_VEL
LIN {X 0,Y 573.257,Z 705.076,A -85,B 0,C 180,E1 -2144.01,E2 -2144.01} C_VEL
LIN {X 0,Y 573.229,Z 705.076,A -85,B 0,C 180,E1 -2146.529,E2 -2146.529} C_VEL
LIN {X 0,Y 573.268,Z 705.072,A -85,B 0,C 180,E1 -2148.745,E2 -2148.745} C_VEL
LIN {X 0,Y 573.283,Z 705.077,A -85,B 0,C 180,E1 -2151.54,E2 -2151.54} C_VEL
LIN {X 0,Y 573.282,Z 705.07,A -85,B 0,C 180,E1 -2154.372,E2 -2154.372} C_VEL
LIN {X 0,Y 573.313,Z 705.074,A -85,B 0,C 180,E1 -2157.892,E2 -2157.892} C_VEL
LIN {X 0,Y 573.332,Z 705.062,A -85,B 0,C 180,E1 -2160.702,E2 -2160.702} C_VEL
LIN {X 0,Y 573.307,Z 705.064,A -85,B 0,C 180,E1 -2162.811,E2 -2162.811} C_VEL
LIN {X 0,Y 573.286,Z 705.073,A -85,B 0,C 180,E1 -2165.628,E2 -2165.628} C_VEL
LIN {X 0,Y 573.267,Z 705.077,A -85,B 0,C 180,E1 -2167.75,E2 -2167.75} C_VEL
LIN {X 0,Y 573.271,Z 705.072,A -85,B 0,C 180,E1 -2170.597,E2 -2170.597} C_VEL
LIN {X 0,Y 573.266,Z 705.071,A -85,B 0,C 180,E1 -2172.749,E2 -2172.749} C_VEL
LIN {X 0,Y 573.239,Z 705.073,A -85,B 0,C 180,E1 -2174.92,E2 -2174.92} C_VEL
LIN {X 0,Y 573.247,Z 705.078,A -85,B 0,C 180,E1 -2177.848,E2 -2177.848} C_VEL
LIN {X 0,Y 573.247,Z 705.082,A -85,B 0,C 180,E1 -2180.077,E2 -2180.077} C_VEL
LIN {X 0,Y 573.238,Z 705.083,A -85,B 0,C 180,E1 -2182.338,E2 -2182.338} C_VEL
LIN {X 0,Y 573.252,Z 705.072,A -85,B 0,C 180,E1 -2185.41,E2 -2185.41} C_VEL
LIN {X 0,Y 573.256,Z 705.077,A -85,B 0,C 180,E1 -2188.029,E2 -2188.029} C_VEL
LIN {X 0,Y 573.233,Z 705.077,A -85,B 0,C 180,E1 -2190.882,E2 -2190.882} C_VEL
LIN {X 0,Y 573.267,Z 705.07,A -85,B 0,C 180,E1 -2193.524,E2 -2193.524} C_VEL
LIN {X 0,Y 573.219,Z 705.08,A -85,B 0,C 180,E1 -2196.051,E2 -2196.051} C_VEL
LIN {X 0,Y 573.251,Z 705.081,A -85,B 0,C 180,E1 -2198.701,E2 -2198.701} C_VEL
LIN {X 0,Y 573.234,Z 705.076,A -85,B 0,C 180,E1 -2201.457,E2 -2201.457} C_VEL
LIN {X 0,Y 573.239,Z 705.08,A -85,B 0,C 180,E1 -2204.333,E2 -2204.333} C_VEL
LIN {X 0,Y 573.245,Z 705.076,A -85,B 0,C 180,E1 -2207.358,E2 -2207.358} C_VEL
LIN {X 0,Y 573.244,Z 705.081,A -85,B 0,C 180,E1 -2210.392,E2 -2210.392} C_VEL
LIN {X 0,Y 573.303,Z 705.232,A -85,B 0,C 180,E1 -2213.191,E2 -2213.191} C_VEL
LIN {X 0,Y 574.185,Z 711.228,A -85,B 0,C 180,E1 -2214.451,E2 -2214.451} C_VEL
LIN {X 0,Y 574.283,Z 727.519,A -85,B 0,C 180,E1 -2217.609,E2 -2217.609} C_VEL
LIN {X 0,Y 574.276,Z 737.103,A -85,B 0,C 180,E1 -2219.477,E2 -2219.477} C_VEL
LIN {X 0,Y 574.039,Z 750.798,A -85,B 0,C 180,E1 -2222.274,E2 -2222.274} C_VEL
LIN {X 0,Y 573.842,Z 764.985,A -85,B 0,C 180,E1 -2225.103,E2 -2225.103} C_VEL
LIN {X 0,Y 573.658,Z 778.188,A -85,B 0,C 180,E1 -2227.679,E2 -2227.679} C_VEL
LIN {X 0,Y 573.514,Z 791.885,A -85,B 0,C 180,E1 -2230.306,E2 -2230.306} C_VEL
LIN {X 0,Y 573.39,Z 805.88,A -85,B 0,C 180,E1 -2232.949,E2 -2232.949} C_VEL
LIN {X 0,Y 573.247,Z 821.229,A -85,B 0,C 180,E1 -2235.806,E2 -2235.806} C_VEL
LIN {X 0,Y 573.191,Z 830.11,A -85,B 0,C 180,E1 -2237.444,E2 -2237.444} C_VEL
LIN {X 0,Y 573.897,Z 835.939,A -85,B 0,C 180,E1 -2237.558,E2 -2237.558} C_VEL
LIN {X 0,Y 573.809,Z 849.214,A -85,B 0,C 180,E1 -2237.87,E2 -2237.87} C_VEL
LIN {X 0,Y 573.717,Z 861.368,A -85,B 0,C 180,E1 -2238.294,E2 -2238.294} C_VEL
LIN {X 0,Y 573.575,Z 873.713,A -85,B 0,C 180,E1 -2238.878,E2 -2238.878} C_VEL
LIN {X 0,Y 573.437,Z 885.2,A -85,B 0,C 180,E1 -2239.585,E2 -2239.585} C_VEL
LIN {X 0,Y 573.332,Z 895.596,A -85,B 0,C 180,E1 -2240.385,E2 -2240.385} C_VEL
LIN {X 0,Y 573.241,Z 904.111,A -85,B 0,C 180,E1 -2241.184,E2 -2241.184} C_VEL
LIN {X 0,Y 573.161,Z 911.959,A -85,B 0,C 180,E1 -2242.071,E2 -2242.071} C_VEL
LIN {X 0,Y 573.073,Z 919.953,A -85,B 0,C 180,E1 -2243.185,E2 -2243.185} C_VEL
LIN {X 0,Y 573.07,Z 926.68,A -85,B 0,C 180,E1 -2244.37,E2 -2244.37} C_VEL
LIN {X 0,Y 573.029,Z 931.371,A -85,B 0,C 180,E1 -2245.427,E2 -2245.427} C_VEL
LIN {X 0,Y 573.023,Z 934.956,A -85,B 0,C 180,E1 -2246.484,E2 -2246.484} C_VEL
LIN {X 0,Y 572.959,Z 936.808,A -85,B 0,C 180,E1 -2247.188,E2 -2247.188} C_VEL
LIN {X 0,Y 572.937,Z 938.2,A -85,B 0,C 180,E1 -2247.891,E2 -2247.891} C_VEL
LIN {X 0,Y 572.941,Z 939.784,A -85,B 0,C 180,E1 -2249.297,E2 -2249.297} C_VEL
LIN {X 0,Y 572.938,Z 940,A -85,B 0,C 180,E1 -2250,E2 -2250} C_VEL
LIN {X 0,Y 572.946,Z 939.185,A -85,B 0,C 180,E1 -2251.406,E2 -2251.406} C_VEL
LIN {X 0,Y 572.937,Z 938.201,A -85,B 0,C 180,E1 -2252.109,E2 -2252.109} C_VEL
LIN {X 0,Y 572.959,Z 936.81,A -85,B 0,C 180,E1 -2252.812,E2 -2252.812} C_VEL
LIN {X 0,Y 573.014,Z 933.896,A -85,B 0,C 180,E1 -2253.868,E2 -2253.868} C_VEL
LIN {X 0,Y 572.963,Z 929.95,A -85,B 0,C 180,E1 -2254.926,E2 -2254.926} C_VEL
LIN {X 0,Y 573.064,Z 923.878,A -85,B 0,C 180,E1 -2256.16,E2 -2256.16} C_VEL
LIN {X 0,Y 573.119,Z 917.237,A -85,B 0,C 180,E1 -2257.221,E2 -2257.221} C_VEL
LIN {X 0,Y 573.201,Z 908.99,A -85,B 0,C 180,E1 -2258.283,E2 -2258.283} C_VEL
LIN {X 0,Y 573.287,Z 900.538,A -85,B 0,C 180,E1 -2259.17,E2 -2259.17} C_VEL
LIN {X 0,Y 573.419,Z 890.096,A -85,B 0,C 180,E1 -2260.058,E2 -2260.058} C_VEL
LIN {X 0,Y 573.541,Z 878.512,A -85,B 0,C 180,E1 -2260.848,E2 -2260.848} C_VEL
LIN {X 0,Y 573.64,Z 866.881,A -85,B 0,C 180,E1 -2261.466,E2 -2261.466} C_VEL
LIN {X 0,Y 573.751,Z 854.175,A -85,B 0,C 180,E1 -2261.974,E2 -2261.974} C_VEL
LIN {X 0,Y 573.853,Z 841.521,A -85,B 0,C 180,E1 -2262.331,E2 -2262.331} C_VEL
LIN {X 0,Y 573.672,Z 833.111,A -85,B 0,C 180,E1 -2262.492,E2 -2262.492} C_VEL
LIN {X 0,Y 573.193,Z 830.034,A -85,B 0,C 180,E1 -2262.57,E2 -2262.57} C_VEL
LIN {X 0,Y 573.313,Z 815.361,A -85,B 0,C 180,E1 -2265.281,E2 -2265.281} C_VEL
LIN {X 0,Y 573.458,Z 799.71,A -85,B 0,C 180,E1 -2268.211,E2 -2268.211} C_VEL
LIN {X 0,Y 573.615,Z 784.54,A -85,B 0,C 180,E1 -2271.096,E2 -2271.096} C_VEL
LIN {X 0,Y 573.776,Z 770.363,A -85,B 0,C 180,E1 -2273.841,E2 -2273.841} C_VEL
LIN {X 0,Y 573.961,Z 756.222,A -85,B 0,C 180,E1 -2276.637,E2 -2276.637} C_VEL
LIN {X 0,Y 574.186,Z 741.328,A -85,B 0,C 180,E1 -2279.653,E2 -2279.653} C_VEL
LIN {X 0,Y 574.274,Z 730.979,A -85,B 0,C 180,E1 -2281.752,E2 -2281.752} C_VEL
LIN {X 0,Y 574.337,Z 718.404,A -85,B 0,C 180,E1 -2284.256,E2 -2284.256} C_VEL
LIN {X 0,Y 574.306,Z 710.188,A -85,B 0,C 180,E1 -2285.972,E2 -2285.972} C_VEL
LIN {X 0,Y 573.257,Z 705.082,A -85,B 0,C 180,E1 -2287.166,E2 -2287.166} C_VEL
LIN {X 0,Y 573.245,Z 705.08,A -85,B 0,C 180,E1 -2289.607,E2 -2289.607} C_VEL
LIN {X 0,Y 573.244,Z 705.076,A -85,B 0,C 180,E1 -2292.642,E2 -2292.642} C_VEL
LIN {X 0,Y 573.238,Z 705.079,A -85,B 0,C 180,E1 -2295.667,E2 -2295.667} C_VEL
LIN {X 0,Y 573.233,Z 705.075,A -85,B 0,C 180,E1 -2298.543,E2 -2298.543} C_VEL
LIN {X 0,Y 573.251,Z 705.08,A -85,B 0,C 180,E1 -2301.299,E2 -2301.299} C_VEL
LIN {X 0,Y 573.217,Z 705.079,A -85,B 0,C 180,E1 -2304.018,E2 -2304.018} C_VEL
LIN {X 0,Y 573.289,Z 705.067,A -85,B 0,C 180,E1 -2306.519,E2 -2306.519} C_VEL
LIN {X 0,Y 573.231,Z 705.078,A -85,B 0,C 180,E1 -2309.118,E2 -2309.118} C_VEL
LIN {X 0,Y 573.255,Z 705.077,A -85,B 0,C 180,E1 -2311.971,E2 -2311.971} C_VEL
LIN {X 0,Y 573.254,Z 705.072,A -85,B 0,C 180,E1 -2314.59,E2 -2314.59} C_VEL
LIN {X 0,Y 573.237,Z 705.083,A -85,B 0,C 180,E1 -2317.662,E2 -2317.662} C_VEL
LIN {X 0,Y 573.269,Z 705.07,A -85,B 0,C 180,E1 -2320.67,E2 -2320.67} C_VEL
LIN {X 0,Y 573.253,Z 705.079,A -85,B 0,C 180,E1 -2323.622,E2 -2323.622} C_VEL
LIN {X 0,Y 573.274,Z 705.079,A -85,B 0,C 180,E1 -2325.807,E2 -2325.807} C_VEL
LIN {X 0,Y 573.267,Z 705.071,A -85,B 0,C 180,E1 -2328.745,E2 -2328.745} C_VEL
LIN {X 0,Y 573.285,Z 705.072,A -85,B 0,C 180,E1 -2331.541,E2 -2331.541} C_VEL
LIN {X 0,Y 573.248,Z 705.078,A -85,B 0,C 180,E1 -2333.665,E2 -2333.665} C_VEL
LIN {X 0,Y 573.231,Z 705.081,A -85,B 0,C 180,E1 -2335.781,E2 -2335.781} C_VEL
LIN {X 0,Y 573.315,Z 705.072,A -85,B 0,C 180,E1 -2337.893,E2 -2337.893} C_VEL
LIN {X 0,Y 573.32,Z 705.066,A -85,B 0,C 180,E1 -2340.702,E2 -2340.702} C_VEL
LIN {X 0,Y 573.293,Z 705.069,A -85,B 0,C 180,E1 -2342.811,E2 -2342.811} C_VEL
LIN {X 0,Y 573.28,Z 705.071,A -85,B 0,C 180,E1 -2345.628,E2 -2345.628} C_VEL
LIN {X 0,Y 573.281,Z 705.076,A -85,B 0,C 180,E1 -2348.46,E2 -2348.46} C_VEL
LIN {X 0,Y 573.276,Z 705.07,A -85,B 0,C 180,E1 -2351.312,E2 -2351.312} C_VEL
LIN {X 0,Y 573.271,Z 705.08,A -85,B 0,C 180,E1 -2354.419,E2 -2354.419} C_VEL
LIN {X 0,Y 573.249,Z 705.074,A -85,B 0,C 180,E1 -2357.112,E2 -2357.112} C_VEL
LIN {X 0,Y 573.24,Z 705.078,A -85,B 0,C 180,E1 -2360.077,E2 -2360.077} C_VEL
LIN {X 0,Y 573.231,Z 705.083,A -85,B 0,C 180,E1 -2362.338,E2 -2362.338} C_VEL
LIN {X 0,Y 573.214,Z 705.082,A -85,B 0,C 180,E1 -2364.367,E2 -2364.367} C_VEL
LIN {X 0,Y 572.568,Z 705.168,A -85,B 0,C 180,E1 -2364.953,E2 -2364.953} C_VEL
LIN {X 0,Y 569.716,Z 705.523,A -85,B 0,C 180,E1 -2365.904,E2 -2365.904} C_VEL
LIN {X 0,Y 567.291,Z 705.825,A -85,B 0,C 180,E1 -2366.67,E2 -2366.67} C_VEL
LIN {X 0,Y 566.248,Z 705.947,A -85,B 0,C 180,E1 -2367.261,E2 -2367.261} C_VEL
LIN {X 0,Y 566.163,Z 705.956,A -85,B 0,C 180,E1 -2367.461,E2 -2367.461} C_VEL
LIN {X 0,Y 566.17,Z 705.955,A -85,B 0,C 180,E1 -2369.771,E2 -2369.771} C_VEL
